// mobject-collections/_Internal/Events/Collection/CollectionEvent
{attribute 'linkalways'} 
{attribute 'no_explicit_call' := 'This FB is a CLASS and must be accessed using methods or properties'}
{attribute 'enable_dynamic_creation'}
FUNCTION_BLOCK ABSTRACT CollectionEvent EXTENDS Disposable
VAR
	_target : I_Collection;
END_VAR

METHOD FB_init : BOOL
VAR_INPUT
	bInitRetains : BOOL; // if TRUE, the retain variables are initialized (warm start / cold start)
	bInCopyCode : BOOL;  // if TRUE, the instance afterwards gets moved into the copy code (online change)
	Target : I_Collection;
END_VAR
This^._target := Target;
END_METHOD

PROPERTY PUBLIC Target : I_Collection
GET
PUBLIC
Target := _target;
END_GET
END_PROPERTY

END_FUNCTION_BLOCK

// mobject-collections/Interfaces/Collections/Events/I_CollectionChangedEvent
INTERFACE I_CollectionChangedEvent EXTENDS I_Event

PROPERTY PUBLIC Target : I_Collection
GET
END_GET
END_PROPERTY

END_INTERFACE

// mobject-collections/_Internal/Events/Collection/CollectionDisposedEvent
{attribute 'linkalways'} 
{attribute 'no_explicit_call' := 'This FB is a CLASS and must be accessed using methods or properties'}
{attribute 'enable_dynamic_creation'}
FUNCTION_BLOCK CollectionDisposedEvent EXTENDS CollectionEvent IMPLEMENTS I_CollectionDisposedEvent

END_FUNCTION_BLOCK

// mobject-collections/Interfaces/Collections/Events/I_CollectionDisposedEvent
INTERFACE I_CollectionDisposedEvent EXTENDS I_Event

PROPERTY PUBLIC Target : I_Collection
GET
END_GET
END_PROPERTY

END_INTERFACE

// mobject-collections/_Internal/Events/KeyValueCollection/KeyValueCollectionChangedEvent
{attribute 'linkalways'} 
{attribute 'no_explicit_call' := 'This FB is a CLASS and must be accessed using methods or properties'}
{attribute 'enable_dynamic_creation'}
FUNCTION_BLOCK KeyValueCollectionChangedEvent EXTENDS KeyValueCollectionEvent IMPLEMENTS I_KeyValueCollectionChangedEvent

END_FUNCTION_BLOCK

// mobject-collections/_Internal/Events/KeyValueCollection/KeyValueCollectionEvent
{attribute 'linkalways'} 
{attribute 'no_explicit_call' := 'This FB is a CLASS and must be accessed using methods or properties'}
{attribute 'enable_dynamic_creation'}
FUNCTION_BLOCK ABSTRACT KeyValueCollectionEvent EXTENDS Disposable
VAR
	_target : I_KeyValueCollection;
END_VAR

METHOD FB_init : BOOL
VAR_INPUT
	bInitRetains : BOOL; // if TRUE, the retain variables are initialized (warm start / cold start)
	bInCopyCode : BOOL;  // if TRUE, the instance afterwards gets moved into the copy code (online change)
	Target : I_KeyValueCollection;
END_VAR
This^._target := Target;
END_METHOD

PROPERTY PUBLIC Target : I_KeyValueCollection
GET
PUBLIC
Target := _target;
END_GET
END_PROPERTY

END_FUNCTION_BLOCK

// mobject-collections/_Internal/Events/KeyValueCollection/KeyValueCollectionDisposedEvent
{attribute 'linkalways'} 
{attribute 'no_explicit_call' := 'This FB is a CLASS and must be accessed using methods or properties'}
{attribute 'enable_dynamic_creation'}
FUNCTION_BLOCK KeyValueCollectionDisposedEvent EXTENDS KeyValueCollectionEvent IMPLEMENTS I_KeyValueCollectionDisposedEvent

END_FUNCTION_BLOCK

// mobject-collections/_Internal/LinkedList/Enumerator/LinkedListForwardEnumerator
{attribute 'linkalways'} 
{attribute 'no_explicit_call' := 'This FB is a CLASS and must be accessed using methods or properties'}
{attribute 'enable_dynamic_creation'}
FUNCTION_BLOCK LinkedListForwardEnumerator EXTENDS Disposable IMPLEMENTS I_ForwardEnumerator, I_EventHandler
VAR
	parent : I_LinkedList;
	currentNode : I_LinkedListNode;
	moveNextCalled : BOOL := FALSE;
	invalid : BOOL := FALSE; 
END_VAR

METHOD FB_init : BOOL
VAR_INPUT
	bInitRetains : BOOL; // if TRUE, the retain variables are initialized (warm start / cold start)
	bInCopyCode : BOOL;  // if TRUE, the instance afterwards gets moved into the copy code (online change)
	Parent : I_LinkedList;
END_VAR
Parent.OnEvent('OnChanged',THIS^);
Parent.OnEvent('OnDisposed',THIS^);
this^.parent := Parent;
END_METHOD

METHOD FB_exit : BOOL
VAR_INPUT
	bInCopyCode : BOOL; // if TRUE, the exit method is called for exiting an instance that is copied afterwards (online change).
END_VAR
IF bInCopyCode THEN
	RETURN;
END_IF

IF parent = 0 THEN
	RETURN;
END_IF

parent.OffEvent('OnChanged',THIS^);
parent.OffEvent('OnDisposed',THIS^);
END_METHOD

METHOD PUBLIC HandleEvent
VAR_INPUT
	Event : I_Event;
END_VAR
VAR
	changedEvent : I_CollectionChangedEvent;
	disposedEvent : I_CollectionDisposedEvent;
END_VAR
IF __QUERYINTERFACE(Event, changedEvent) THEN
	invalid := TRUE;
	currentNode := 0;
ELSIF __QUERYINTERFACE(Event, disposedEvent) THEN
	parent := 0;
	Dispose();
END_IF
END_METHOD

PROPERTY PUBLIC IsValid : BOOL
GET
PUBLIC
IsValid := (not invalid and parent <> 0);
END_GET
END_PROPERTY

METHOD PUBLIC MoveNext : BOOL
IF invalid THEN
	RETURN;
END_IF

IF NOT moveNextCalled THEN
	moveNextCalled := TRUE;	
	currentNode := parent.First;
	MoveNext := currentNode <> 0;
	RETURN;
END_IF

IF currentNode = 0 THEN
	RETURN;
END_IF

if currentNode.Next <> 0 then
	currentNode := currentNode.Next;
	MoveNext := TRUE;	
	RETURN;
END_IF
END_METHOD

METHOD Reset
VAR_INPUT
END_VAR
moveNextCalled := FALSE;
currentNode := 0;
END_METHOD

METHOD PUBLIC TryGet : BOOL;
VAR_INPUT
	Destination : ANY;
END_VAR
IF currentNode <> 0 THEN
	TryGet := currentNode.TryGet(Destination);
END_IF
END_METHOD

METHOD PUBLIC TryGetTo : BOOL;
VAR_INPUT
	DestinationAddress : PVOID;
	DestinationSize : UDINT;
END_VAR
IF currentNode <> 0 THEN
	TryGetTo := currentNode.TryGetTo(DestinationAddress,DestinationSize);
END_IF
END_METHOD

END_FUNCTION_BLOCK

// mobject-collections/Interfaces/Collections/I_LinkedList
INTERFACE I_LinkedList EXTENDS I_Collection

METHOD PUBLIC AddAfter
VAR_INPUT
	After : I_LinkedListNode;
	Value : ANY;
END_VAR
END_METHOD

METHOD PUBLIC AddBefore
VAR_INPUT
	Before : I_LinkedListNode;
	Value : ANY;
END_VAR
END_METHOD

METHOD PUBLIC AddFirst
VAR_INPUT
	Value : ANY;
END_VAR
END_METHOD

METHOD PUBLIC AddLast
VAR_INPUT
	Value : ANY;
END_VAR
END_METHOD

METHOD PUBLIC Find : I_LinkedListNode
VAR_INPUT
	Value : ANY;
END_VAR
END_METHOD

METHOD PUBLIC FindLast : I_LinkedListNode
VAR_INPUT
	Value : ANY;
END_VAR
END_METHOD

PROPERTY PUBLIC First : I_LinkedListNode
GET
END_GET
END_PROPERTY

PROPERTY PUBLIC Last : I_LinkedListNode
GET
END_GET
END_PROPERTY

METHOD PUBLIC Remove
VAR_INPUT
	Value : ANY;
END_VAR
END_METHOD

METHOD PUBLIC RemoveFirst
END_METHOD

METHOD PUBLIC RemoveLast
END_METHOD

END_INTERFACE

// mobject-collections/Interfaces/Collections/Nodes/I_LinkedListNode
INTERFACE I_LinkedListNode EXTENDS I_CollectionNode

PROPERTY PUBLIC Next : I_LinkedListNode
GET
END_GET
SET
END_SET
END_PROPERTY

PROPERTY PUBLIC Previous : I_LinkedListNode
GET
END_GET
SET
END_SET
END_PROPERTY

END_INTERFACE

// mobject-collections/_Internal/LinkedList/Node/LinkedListNode
{attribute 'linkalways'} 
{attribute 'no_explicit_call' := 'This FB is a CLASS and must be accessed using methods or properties'}
{attribute 'enable_dynamic_creation'}
FUNCTION_BLOCK LinkedListNode EXTENDS Disposable IMPLEMENTS I_LinkedListNode
VAR
	pBuffer : POINTER TO BYTE;
	bufferSize : UDINT;
	_previous : I_LinkedListNode;
	_next : I_LinkedListNode;
END_VAR

METHOD FB_init : BOOL
VAR_INPUT
	bInitRetains : BOOL; // if TRUE, the retain variables are initialized (warm start / cold start)
	bInCopyCode : BOOL;  // if TRUE, the instance afterwards gets moved into the copy code (online change)
	Source : ANY;
END_VAR
CreateBuffer(DINT_TO_UDINT(Source.diSize));
CopySourceToBuffer(Source.pValue);
END_METHOD

METHOD FB_exit : BOOL
VAR_INPUT
	bInCopyCode : BOOL; // if TRUE, the exit method is called for exiting an instance that is copied afterwards (online change).
END_VAR
IF bInCopyCode THEN
	RETURN;
END_IF

DestroyBuffer();
END_METHOD

METHOD PRIVATE CopyBufferToDestination
VAR_INPUT
	DestinationAddress : PVOID;
END_VAR
MEMCPY(DestinationAddress, pBuffer, bufferSize);
END_METHOD

METHOD PRIVATE CopySourceToBuffer
VAR_INPUT
	SourceAddress : PVOID;
END_VAR
MEMCPY(pBuffer, SourceAddress, bufferSize);
END_METHOD

METHOD PRIVATE CreateBuffer
VAR_INPUT
	SizeInBytes : UDINT;
END_VAR
bufferSize := SizeInBytes;
pBuffer := __NEW(BYTE, SizeInBytes);
END_METHOD

METHOD PRIVATE DestroyBuffer
IF pBuffer = 0 THEN
	RETURN;
END_IF

__DELETE(pBuffer);
bufferSize := 0;
END_METHOD

PROPERTY PUBLIC DataSize : UDINT
GET
PUBLIC
DataSize := bufferSize;
END_GET
END_PROPERTY

METHOD PUBLIC Equals : BOOL
VAR_INPUT
	Symbol : ANY;
END_VAR
IF pBuffer = 0 THEN
	RETURN;
END_IF

IF bufferSize <> DINT_TO_UDINT(Symbol.diSize) THEN
	RETURN;
END_IF

Equals := MEMCMP(Symbol.pValue, pBuffer, bufferSize) = 0;
END_METHOD

PROPERTY PUBLIC Next : I_LinkedListNode
GET
PUBLIC
Next := _next;
END_GET
SET
PUBLIC
_next := Next;
END_SET
END_PROPERTY

PROPERTY PUBLIC Previous : I_LinkedListNode
GET
PUBLIC
Previous := _previous;
END_GET
SET
PUBLIC
_previous := Previous;
END_SET
END_PROPERTY

METHOD PUBLIC TryGet : BOOL;
VAR_INPUT
	Destination : ANY;
END_VAR
TryGet := TryGetTo(Destination.pValue, DINT_TO_UDINT(Destination.diSize));
END_METHOD

METHOD PUBLIC TryGetTo : BOOL;
VAR_INPUT
	DestinationAddress : PVOID;
	DestinationSize : UDINT;
END_VAR
IF pBuffer = 0 THEN
	RETURN;
END_IF

IF bufferSize <> DestinationSize THEN
	RETURN;
END_IF

CopyBufferToDestination(DestinationAddress);
TryGetTo := TRUE;
END_METHOD

END_FUNCTION_BLOCK

// mobject-collections/_Internal/OrderedDictionary/Enumerator/OrderedDictionaryForwardEnumerator
{attribute 'linkalways'} 
{attribute 'no_explicit_call' := 'This FB is a CLASS and must be accessed using methods or properties'}
{attribute 'enable_dynamic_creation'}
FUNCTION_BLOCK OrderedDictionaryForwardEnumerator EXTENDS Disposable IMPLEMENTS I_KeyValueForwardEnumerator, I_EventHandler
VAR
	parent : I_Dictionary;
	nodes : I_Collection;
	collectionEnumerator : I_ForwardEnumerator;
	currentNode : I_OrderedDictionaryTreeNode;
	moveNextCalled : BOOL := FALSE;
	invalid : BOOL := FALSE; 
END_VAR

METHOD FB_init : BOOL
VAR_INPUT
	bInitRetains : BOOL; // if TRUE, the retain variables are initialized (warm start / cold start)
	bInCopyCode : BOOL;  // if TRUE, the instance afterwards gets moved into the copy code (online change)
	Parent : I_Dictionary;
	Nodes : I_Collection;
END_VAR
Parent.OnEvent('OnChanged',THIS^);
Parent.OnEvent('OnDisposed',THIS^);
THIS^.parent := Parent;
THIS^.nodes := Nodes;
THIS^.collectionEnumerator := Nodes.GetEnumerator();
END_METHOD

METHOD FB_exit : BOOL
VAR_INPUT
	bInCopyCode : BOOL; // if TRUE, the exit method is called for exiting an instance that is copied afterwards (online change).
END_VAR
IF bInCopyCode THEN
	RETURN;
END_IF

collectionEnumerator.Dispose();
nodes.Dispose();

IF parent = 0 THEN
	RETURN;
END_IF

parent.OffEvent('OnChanged',THIS^);
parent.OffEvent('OnDisposed',THIS^);
END_METHOD

METHOD PUBLIC HandleEvent
VAR_INPUT
	Event : I_Event;
END_VAR
VAR
	changedEvent : I_KeyValueCollectionChangedEvent;
	disposedEvent : I_KeyValueCollectionDisposedEvent;
END_VAR
IF __QUERYINTERFACE(Event, changedEvent) THEN
	invalid := TRUE;
	currentNode := 0;
ELSIF __QUERYINTERFACE(Event, disposedEvent) THEN
	parent := 0;	
	Dispose();
END_IF
END_METHOD

PROPERTY PUBLIC IsValid : BOOL
GET
PUBLIC
IsValid := (not invalid and parent <> 0);
END_GET
END_PROPERTY

PROPERTY PUBLIC Key : T_MAXSTRING
GET
IF NOT IsValid THEN
	RETURN;
END_IF

IF currentNode = 0 THEN
	RETURN;
END_IF

Key := currentNode.Key;
END_GET
END_PROPERTY

METHOD PUBLIC MoveNext : BOOL
IF invalid THEN
	RETURN;
END_IF

IF collectionEnumerator.MoveNext() THEN
	collectionEnumerator.TryGet(currentNode);
	MoveNext := TRUE;
END_IF
END_METHOD

METHOD Reset
VAR_INPUT
END_VAR
moveNextCalled := FALSE;
collectionEnumerator.Reset();
END_METHOD

METHOD PUBLIC TryGet : BOOL;
VAR_INPUT
	Destination : ANY;
END_VAR
IF currentNode <> 0 THEN
	TryGet := currentNode.TryGet(Destination);
END_IF
END_METHOD

METHOD PUBLIC TryGetTo : BOOL;
VAR_INPUT
	DestinationAddress : PVOID;
	DestinationSize : UDINT;
END_VAR
IF currentNode <> 0 THEN
	TryGetTo := currentNode.TryGetTo(DestinationAddress,DestinationSize);
END_IF
END_METHOD

END_FUNCTION_BLOCK

// mobject-collections/Interfaces/KeyValueCollections/Nodes/I_OrderedDictionaryTreeNode
INTERFACE I_OrderedDictionaryTreeNode EXTENDS I_CollectionNode

METHOD PUBLIC DeepCopy
VAR_INPUT
	Node : I_OrderedDictionaryTreeNode;
END_VAR
END_METHOD

PROPERTY PUBLIC Height : DINT
GET
END_GET
SET
END_SET
END_PROPERTY

PROPERTY PUBLIC Key : T_MAXSTRING
GET
END_GET
END_PROPERTY

PROPERTY PUBLIC Left : I_OrderedDictionaryTreeNode
GET
END_GET
SET
END_SET
END_PROPERTY

PROPERTY PUBLIC Next : I_OrderedDictionaryTreeNode
GET
END_GET
SET
END_SET
END_PROPERTY

PROPERTY PUBLIC NodeBufferPointer : Pointer To Byte
GET
END_GET
END_PROPERTY

PROPERTY PUBLIC NodeBufferSize : UDINT
GET
END_GET
END_PROPERTY

PROPERTY PUBLIC Previous : I_OrderedDictionaryTreeNode
GET
END_GET
SET
END_SET
END_PROPERTY

METHOD Reinitialize
VAR_INPUT
	Key : T_MAXSTRING;
	Source : ANY;
END_VAR
END_METHOD

PROPERTY PUBLIC Right : I_OrderedDictionaryTreeNode
GET
END_GET
SET
END_SET
END_PROPERTY

END_INTERFACE

// mobject-collections/_Internal/OrderedDictionary/Node/OrderedDictionaryTreeNode
{attribute 'linkalways'} 
{attribute 'no_explicit_call' := 'This FB is a CLASS and must be accessed using methods or properties'}
{attribute 'enable_dynamic_creation'}
FUNCTION_BLOCK OrderedDictionaryTreeNode EXTENDS Disposable IMPLEMENTS I_OrderedDictionaryTreeNode
VAR
	_key : T_MAXSTRING;
	pBuffer : POINTER TO BYTE;
	bufferSize : UDINT;
    _height : DINT;
    _left : I_OrderedDictionaryTreeNode;
    _right : I_OrderedDictionaryTreeNode;
	_next : I_OrderedDictionaryTreeNode;
    _previous : I_OrderedDictionaryTreeNode;
END_VAR

METHOD FB_init : BOOL
VAR_INPUT
	bInitRetains : BOOL; // if TRUE, the retain variables are initialized (warm start / cold start)
	bInCopyCode : BOOL;  // if TRUE, the instance afterwards gets moved into the copy code (online change)
	NodeKey : T_MAXSTRING;
	NodeSource : ANY;
END_VAR
_key := NodeKey;
CreateBuffer(DINT_TO_UDINT(NodeSource.diSize));
CopySourceToBuffer(NodeSource.pValue);
END_METHOD

METHOD FB_exit : BOOL
VAR_INPUT
	bInCopyCode : BOOL; // if TRUE, the exit method is called for exiting an instance that is copied afterwards (online change).
END_VAR
IF bInCopyCode THEN
	RETURN;
END_IF

DestroyBuffer();
END_METHOD

METHOD PRIVATE CopyBufferToDestination
VAR_INPUT
	DestinationAddress : PVOID;
END_VAR
MEMCPY(DestinationAddress, pBuffer, bufferSize);
END_METHOD

METHOD PRIVATE CopySourceToBuffer
VAR_INPUT
	SourceAddress : PVOID;
END_VAR
MEMCPY(pBuffer, SourceAddress, bufferSize);
END_METHOD

METHOD PRIVATE CreateBuffer
VAR_INPUT
	SizeInBytes : UDINT;
END_VAR
bufferSize := SizeInBytes;
pBuffer := __NEW(BYTE, SizeInBytes);
END_METHOD

METHOD PRIVATE DestroyBuffer
VAR_INPUT
END_VAR
IF pBuffer = 0 THEN
	RETURN;
END_IF

__DELETE(pBuffer);
bufferSize := 0;
END_METHOD

PROPERTY PUBLIC DataSize : UDINT
GET
DataSize := bufferSize;
END_GET
END_PROPERTY

METHOD PUBLIC DeepCopy
VAR_INPUT
	Node : I_OrderedDictionaryTreeNode;
END_VAR
DestroyBuffer();
CreateBuffer(Node.NodeBufferSize);
CopySourceToBuffer(Node.NodeBufferPointer);
_key := Node.Key;
_previous := Node.Previous;
_next := Node.Next;
END_METHOD

METHOD PUBLIC Equals : BOOL
VAR_INPUT
	Symbol : ANY;
END_VAR
IF pBuffer = 0 THEN
	RETURN;
END_IF

IF bufferSize <> DINT_TO_UDINT(symbol.diSize) THEN
	RETURN;
END_IF

Equals := MEMCMP(Symbol.pValue, pBuffer, bufferSize) = 0;
END_METHOD

PROPERTY PUBLIC Height : DINT
GET
Height := _height;
END_GET
SET
PUBLIC 
VAR
END_VAR
_height := Height;
END_SET
END_PROPERTY

PROPERTY PUBLIC Key : T_MAXSTRING
GET
Key := _key;
END_GET
END_PROPERTY

PROPERTY PUBLIC Left : I_OrderedDictionaryTreeNode
GET
Left := _left;
END_GET
SET
_left := Left;
END_SET
END_PROPERTY

PROPERTY PUBLIC Next : I_OrderedDictionaryTreeNode
GET
Next := _next;
END_GET
SET
_next := Next;
END_SET
END_PROPERTY

PROPERTY PUBLIC NodeBufferPointer : Pointer To Byte
GET
NodeBufferPointer := pBuffer;
END_GET
END_PROPERTY

PROPERTY PUBLIC NodeBufferSize : UDINT
GET
NodeBufferSize := bufferSize;
END_GET
END_PROPERTY

PROPERTY PUBLIC Previous : I_OrderedDictionaryTreeNode
GET
Previous := _previous;
END_GET
SET
_previous := Previous;
END_SET
END_PROPERTY

METHOD Reinitialize
VAR_INPUT
	Key : T_MAXSTRING;
	Source : ANY;
END_VAR
_key := Key;

IF pBuffer <> 0 THEN
	DestroyBuffer();
END_IF

CreateBuffer(DINT_TO_UDINT(Source.diSize));
CopySourceToBuffer(Source.pValue);
END_METHOD

PROPERTY PUBLIC Right : I_OrderedDictionaryTreeNode
GET
Right := _right;
END_GET
SET
_right := Right;
END_SET
END_PROPERTY

METHOD TryGet : BOOL
VAR_INPUT
	Destination	: ANY;
END_VAR
TryGet := TryGetTo(Destination.pValue, DINT_TO_UDINT(Destination.diSize));
END_METHOD

METHOD TryGetTo : BOOL
VAR_INPUT
	DestinationAddress : PVOID;
	DestinationSize : UDINT;
END_VAR
IF pBuffer = 0 THEN
	RETURN;
END_IF

IF bufferSize <> DestinationSize THEN
	RETURN;
END_IF

CopyBufferToDestination(DestinationAddress);
TryGetTo := TRUE;
END_METHOD

END_FUNCTION_BLOCK

// mobject-collections/Dictionary/Dictionary
{attribute 'linkalways'} 
{attribute 'no_explicit_call' := 'This FB is a CLASS and must be accessed using methods or properties'}
{attribute 'enable_dynamic_creation'}
FUNCTION_BLOCK Dictionary EXTENDS Disposable IMPLEMENTS I_Dictionary
VAR
	eventEmitter : EventEmitter;
	rootNode : I_DictionaryTreeNode;
END_VAR

METHOD FB_exit : BOOL
VAR_INPUT
	bInCopyCode : BOOL; // if TRUE, the exit method is called for exiting an instance that is copied afterwards (online change).
END_VAR
VAR
END_VAR
IF bInCopyCode THEN
    RETURN;
END_IF

Clear();
EmitDisposedEvent();
END_METHOD

METHOD PRIVATE Balance : I_DictionaryTreeNode
VAR_INPUT
	Node : I_DictionaryTreeNode;
END_VAR
VAR
	balanceFactor : DINT;
END_VAR
balanceFactor := THIS^.GetBalanceFactor(Node);

IF (balanceFactor > 1) THEN
	IF THIS^.GetBalanceFactor(Node.Left) < 0 THEN
		Node.Left := THIS^.LeftRotate(Node.Left);
	END_IF
	Node := RightRotate(Node);
ELSIF (balanceFactor < -1) THEN
	IF THIS^.GetBalanceFactor(Node.Right) > 0 THEN
		Node.Right := RightRotate(Node.Right);
	END_IF
	Node := LeftRotate(Node);
END_IF

Balance := Node;
END_METHOD

METHOD PRIVATE EmitChangedEvent
VAR
	pDictionaryChangedEvent : POINTER TO KeyValueCollectionChangedEvent;
END_VAR
pDictionaryChangedEvent := __NEW(KeyValueCollectionChangedEvent(Target := THIS^));
eventEmitter.Emit('OnChanged', pDictionaryChangedEvent^);
pDictionaryChangedEvent^.Dispose();
END_METHOD

METHOD PRIVATE EmitDisposedEvent
VAR
	pDictionaryDisposedEvent : POINTER TO KeyValueCollectionDisposedEvent;
END_VAR
pDictionaryDisposedEvent := __NEW(KeyValueCollectionDisposedEvent(Target := THIS^));
eventEmitter.Emit('OnDisposed', pDictionaryDisposedEvent^);
pDictionaryDisposedEvent^.Dispose();
END_METHOD

METHOD PRIVATE FindMinimum : I_DictionaryTreeNode
VAR_INPUT
	Node : I_DictionaryTreeNode;
END_VAR
VAR
	nextNode : I_DictionaryTreeNode;
END_VAR
nextNode := Node;

WHILE (nextNode.left <> 0) DO
      nextNode := nextNode.left;
END_WHILE;

FindMinimum := nextNode;
END_METHOD

METHOD PRIVATE GetBalanceFactor : DINT
VAR_INPUT
	Node : I_DictionaryTreeNode;
END_VAR
IF (Node = 0) THEN
	GetBalanceFactor := 0;
	RETURN;
END_IF

GetBalanceFactor := THIS^.GetHeight(node.left) - THIS^.GetHeight(node.right);
END_METHOD

METHOD PRIVATE GetHeight : DINT
VAR_INPUT
	Node : I_DictionaryTreeNode;
END_VAR
IF Node = 0 THEN
	GetHeight := -1;
	RETURN;
END_IF

GetHeight := Node.Height;
END_METHOD

METHOD PRIVATE LeftRotate : I_DictionaryTreeNode
VAR_INPUT
	X : I_DictionaryTreeNode;
END_VAR
VAR
	y : I_DictionaryTreeNode;
	t2 : I_DictionaryTreeNode;
END_VAR
y := X.right;
t2 := y.left;
y.left := X;
X.right := t2;
THIS^.UpdateHeight(X);
THIS^.UpdateHeight(y);
LeftRotate := y;
END_METHOD

METHOD PRIVATE RecursiveAddKeysInOrderToCollection
VAR_INPUT
	Node : I_DictionaryTreeNode;
	Collection : I_Collection;
END_VAR
VAR
	key : T_MAXSTRING;
END_VAR
IF Node = 0 THEN
	RETURN;
END_IF

THIS^.RecursiveAddKeysInOrderToCollection(Node.Left,Collection);
key := Node.Key;
Collection.AddItem(key);
THIS^.RecursiveAddKeysInOrderToCollection(Node.Right,Collection);
END_METHOD

METHOD PRIVATE RecursiveAddNodesInOrderToCollection
VAR_INPUT
	Node : I_DictionaryTreeNode;
	Collection : I_Collection;
END_VAR
IF Node = 0 THEN
	RETURN;
END_IF

THIS^.RecursiveAddNodesInOrderToCollection(Node.Left,Collection);
Collection.AddItem(Node);
THIS^.RecursiveAddNodesInOrderToCollection(Node.Right,Collection);
END_METHOD

METHOD PRIVATE RecursiveClear
VAR_INPUT
	Node : I_DictionaryTreeNode;
END_VAR
VAR
	thisNodeKey : T_MAXSTRING;
	leftNodeKey : T_MAXSTRING;
	rightNodeKey : T_MAXSTRING;
END_VAR
IF (Node = 0) THEN
	RETURN;
END_IF

thisNodeKey := Node.key;

IF (Node.Left <> 0) THEN
	leftNodeKey := Node.Left.key;
END_IF

IF (Node.Right <> 0) THEN
	rightNodeKey := Node.Right.key;
END_IF


RecursiveClear(Node.Left);
RecursiveClear(Node.Right);
Node.Dispose();
END_METHOD

METHOD PRIVATE RecursiveCountNodes
VAR_INPUT
	Node : I_DictionaryTreeNode;
	Count : REFERENCE TO DINT;
END_VAR
IF Node = 0 THEN
	RETURN;
END_IF

Count := Count + 1;

THIS^.RecursiveCountNodes(Node.Left,Count);
THIS^.RecursiveCountNodes(Node.Right,Count);
END_METHOD

METHOD PRIVATE RecursiveDelete : I_DictionaryTreeNode
VAR_INPUT
	Key : T_MAXSTRING;
	Node : I_DictionaryTreeNode;
END_VAR
VAR
	newNode : I_DictionaryTreeNode; 
	minValueNode : I_DictionaryTreeNode;
	minValueNodeParent : I_DictionaryTreeNode;
	balanceFactor : DINT;
END_VAR
IF (Node = 0) THEN
    RETURN;
END_IF

IF (Key < Node.Key) THEN
    Node.left := THIS^.RecursiveDelete(Key, Node.left);
ELSIF (Key > Node.Key) THEN
    Node.right := THIS^.RecursiveDelete(Key, Node.right);
ELSE
    IF (Node.Left = 0) OR (Node.Right = 0) THEN
        IF (Node.Left = 0) THEN
            newNode := Node.Right;
        ELSE
            newNode := Node.Left;
        END_IF

        Node.Dispose();
        THIS^.updateHeight(newNode);
        RecursiveDelete := THIS^.Balance(newNode);
        RETURN;
    ELSE
        minValueNode := FindMinimum(Node.Right);
        Node.DeepCopy(minValueNode);
        Node.Right := THIS^.RecursiveDelete(minValueNode.Key, Node.Right);	
    END_IF
END_IF

THIS^.updateHeight(Node);
RecursiveDelete := THIS^.Balance(Node);
END_METHOD

METHOD PRIVATE RecursiveFind : I_DictionaryTreeNode
VAR_INPUT
	Key : T_MAXSTRING;
	Node : I_DictionaryTreeNode;
END_VAR
IF (Node = 0) THEN
	RETURN;
END_IF

IF (Key < Node.key) THEN
  RecursiveFind := THIS^.RecursiveFind(key, Node.left);
  RETURN;
ELSIF (key > Node.key) THEN
  RecursiveFind := THIS^.RecursiveFind(key, Node.right);
  RETURN;
ELSE 
  RecursiveFind := Node;
  RETURN;
END_IF
END_METHOD

METHOD PRIVATE RecursiveInsert : I_DictionaryTreeNode
VAR_INPUT
	Key : T_MAXSTRING;
	Value : ANY;
	Node : I_DictionaryTreeNode;
END_VAR
VAR
	pAVLTreeNode : POINTER TO DictionaryTreeNode;
	balanceFactor : DINT;
END_VAR
IF (Node = 0) THEN
	pAVLTreeNode := __NEW(DictionaryTreeNode(NodeKey := Key, NodeSource := Value));
	RecursiveInsert := pAVLTreeNode^;
	RETURN;
END_IF

IF (Key < Node.Key) THEN
	Node.left := THIS^.RecursiveInsert(Key, Value, Node.left);
ELSIF (Key > Node.Key) THEN
	Node.right := THIS^.RecursiveInsert(Key, Value, Node.right);
ELSE
	Node.Reinitialize(Key,Value);
	RecursiveInsert := Node;
END_IF

THIS^.updateHeight(node);

Node := balance(Node);
RecursiveInsert := Node;
END_METHOD

METHOD PRIVATE RightRotate : I_DictionaryTreeNode
VAR_INPUT
	Y : I_DictionaryTreeNode;
END_VAR
VAR
	x : I_DictionaryTreeNode;
	t2 : I_DictionaryTreeNode;
END_VAR
x := Y.left;
t2 := x.right;
x.right := Y;
Y.left := t2;
THIS^.UpdateHeight(Y);
THIS^.UpdateHeight(x);
RightRotate := x;
END_METHOD

METHOD PRIVATE UpdateHeight
VAR_INPUT
	Node : I_DictionaryTreeNode;
END_VAR
IF (Node = 0) THEN
	RETURN;
END_IF

Node.height := 1 + MAX(THIS^.GetHeight(Node.left), THIS^.GetHeight(Node.right));
END_METHOD

METHOD PUBLIC AddOrUpdate
VAR_INPUT
	Key : T_MAXSTRING;
	Value : ANY;
END_VAR
rootNode := THIS^.RecursiveInsert(Key, Value, rootNode);
EmitChangedEvent();
END_METHOD

METHOD PUBLIC Clear
VAR_INPUT
END_VAR
IF rootNode = 0 THEN
	RETURN;
END_IF

THIS^.RecursiveClear(rootNode);
rootNode := 0;
EmitChangedEvent();
END_METHOD

METHOD PUBLIC ContainsKey : BOOL
VAR_INPUT
	Key : T_MAXSTRING;
END_VAR
VAR
	foundNode : I_DictionaryTreeNode;
END_VAR
foundNode := THIS^.RecursiveFind(Key, rootNode);

IF foundNode = 0 THEN
	RETURN;
END_IF

ContainsKey := TRUE;
END_METHOD

PROPERTY PUBLIC Count : DINT
GET
VAR
	NodeCount : DINT;
END_VAR
RecursiveCountNodes(rootNode, NodeCount);
Count := NodeCount;
END_GET
END_PROPERTY

METHOD GetEnumerator : I_ForwardEnumerator
VAR
	pNodeCollection : POINTER TO LinkedList;
	pEnumerator : POINTER TO DictionaryForwardEnumerator;
END_VAR
pNodeCollection := __NEW(LinkedList);
THIS^.RecursiveAddNodesInOrderToCollection(rootNode, pNodeCollection^);

pEnumerator := __NEW(DictionaryForwardEnumerator(Parent := THIS^, Nodes := pNodeCollection^));
GetEnumerator := pEnumerator^;
END_METHOD

METHOD PUBLIC GetKeys : I_Collection
VAR
	pLinkedList : POINTER TO LinkedList;
END_VAR
pLinkedList := __NEW(LinkedList);
THIS^.RecursiveAddKeysInOrderToCollection(rootNode,pLinkedList^);
GetKeys := pLinkedList^;
END_METHOD

METHOD GetKeyValueEnumerator : I_KeyValueForwardEnumerator
VAR
	pNodeCollection : POINTER TO LinkedList;
	pEnumerator : POINTER TO DictionaryForwardEnumerator;
END_VAR
pNodeCollection := __NEW(LinkedList);
THIS^.RecursiveAddNodesInOrderToCollection(rootNode, pNodeCollection^);

pEnumerator := __NEW(DictionaryForwardEnumerator(Parent := THIS^, Nodes := pNodeCollection^));
GetKeyValueEnumerator := pEnumerator^;
END_METHOD

PROPERTY IsEmpty : BOOL
GET
IsEmpty := rootNode = 0;
END_GET
END_PROPERTY

METHOD PUBLIC OffEvent
VAR_INPUT
	EventName : T_MaxString;
	EventHandler : I_EventHandler;
END_VAR
eventEmitter.OffEvent(EventName, EventHandler);
END_METHOD

METHOD PUBLIC OnceEvent
VAR_INPUT
	EventName : T_MaxString;
	EventHandler : I_EventHandler;
END_VAR
eventEmitter.OnceEvent(EventName, EventHandler);
END_METHOD

METHOD PUBLIC OnEvent
VAR_INPUT
	EventName : T_MaxString;
	EventHandler : I_EventHandler;
END_VAR
eventEmitter.OnEvent(EventName, EventHandler);
END_METHOD

METHOD PUBLIC Remove
VAR_INPUT
	Key : T_MAXSTRING;
END_VAR
rootNode := THIS^.RecursiveDelete(Key, rootNode);
EmitChangedEvent();
END_METHOD

METHOD PUBLIC TryAdd : BOOL
VAR_INPUT
	Key : T_MAXSTRING;
	Value : ANY;
END_VAR
IF ContainsKey(Key) THEN
	RETURN;
END_IF
	  
THIS^.AddOrUpdate(Key, Value);
TryAdd := TRUE;
END_METHOD

METHOD PUBLIC TryGetValue : BOOL
VAR_INPUT
	Key : T_MAXSTRING;
	Destination	: ANY;
END_VAR
TryGetValue := TryGetValueTo(Key, Destination.pValue, DINT_TO_UDINT(Destination.diSize));
END_METHOD

METHOD PUBLIC TryGetValueTo : BOOL
VAR_INPUT
	Key : T_MAXSTRING;
	DestinationAddress : PVOID;
	DestinationSize : UDINT;
END_VAR
VAR
	foundNode : I_DictionaryTreeNode;
END_VAR
foundNode := THIS^.RecursiveFind(Key, rootNode);

IF foundNode = 0 THEN
	RETURN;
END_IF

TryGetValueTo := foundNode.TryGetTo(DestinationAddress, DestinationSize);
END_METHOD

END_FUNCTION_BLOCK

// mobject-events/EventEmitter/EventEmitter
{attribute 'linkalways'} 
{attribute 'no_explicit_call' := 'This FB is a CLASS and must be accessed using methods or properties'}
{attribute 'enable_dynamic_creation'}
FUNCTION_BLOCK EventEmitter EXTENDS Disposable IMPLEMENTS I_EventEmitter, I_EventTarget
VAR
	firstEventHandlerItem : I_EventHandlerItem;
END_VAR

METHOD FB_exit : BOOL
VAR_INPUT
	bInCopyCode : BOOL; // if TRUE, the exit method is called for exiting an instance that is copied afterwards (online change).
END_VAR
IF bInCopyCode THEN
	RETURN;
END_IF

DisposeAllEventHandlerItems();
END_METHOD

METHOD PRIVATE DisposeAllEventHandlerItems
VAR_INPUT
END_VAR
WHILE firstEventHandlerItem <> 0 DO
	DisposeEventHandlerItem(firstEventHandlerItem);
END_WHILE
END_METHOD

METHOD PRIVATE DisposeEventHandlerItem
VAR_INPUT
	EventHandlerItem : I_EventHandlerItem;
END_VAR
RemoveEventHandlerItemFromCollection(EventHandlerItem);
EventHandlerItem.Dispose();
END_METHOD

METHOD PRIVATE FindEventHandlerItem : I_EventHandlerItem
VAR_INPUT
	EventName : T_MaxString;
	EventHandler : I_EventHandler;
END_VAR
VAR
	currentEventHandlerItem : I_EventHandlerItem;
END_VAR
currentEventHandlerItem := firstEventHandlerItem;

WHILE currentEventHandlerItem <> 0 DO
	
	IF currentEventHandlerItem.EqualTo(EventName, EventHandler) THEN
		FindEventHandlerItem := currentEventHandlerItem; 
		RETURN;
	END_IF
	
	currentEventHandlerItem := currentEventHandlerItem.Next;

END_WHILE
END_METHOD

METHOD PRIVATE InsertEventHandlerItem
VAR_INPUT
	EventHandlerItem : I_EventHandlerItem;
END_VAR
VAR
	currentEventHandlerItem : I_EventHandlerItem;
END_VAR
IF firstEventHandlerItem = 0 THEN
	firstEventHandlerItem := EventHandlerItem;
	RETURN;
END_IF

currentEventHandlerItem := firstEventHandlerItem;

WHILE currentEventHandlerItem.next <> 0 DO
	currentEventHandlerItem := currentEventHandlerItem.next;
END_WHILE

currentEventHandlerItem.next := EventHandlerItem;
EventHandlerItem.previous := currentEventHandlerItem;
END_METHOD

METHOD PRIVATE RemoveEventHandlerItemFromCollection
VAR_INPUT
	EventHandlerItem : I_EventHandlerItem;
END_VAR
VAR
	previous : I_EventHandlerItem;
	next : I_EventHandlerItem;
END_VAR
IF EventHandlerItem = 0 THEN
	// nothing to remove
	RETURN;
END_IF

IF EventHandlerItem = firstEventHandlerItem AND EventHandlerItem.Next = 0 THEN 
	
	// the item was the only one in the list, as such you just set the first to zero
	firstEventHandlerItem := 0; 
	
ELSIF EventHandlerItem = firstEventHandlerItem THEN 
	
	// the item was the first in the list of many, so make the next item the first and remove 
	// it's "previous" as the first in the item does not have a previous
	firstEventHandlerItem := EventHandlerItem.next; 
	firstEventHandlerItem.Previous := 0;

ELSIF EventHandlerItem.Next <> 0 THEN
	
	// the item is mid list so link it's previous and next together 
	previous := EventHandlerItem.Previous;
	next := EventHandlerItem.Next;
	
	previous.Next := next;
	next.Previous := previous;
	
ELSE 
	
	// the item is at the end so only remove itself from the previous
	previous := EventHandlerItem.Previous;
	previous.Next := 0;

END_IF
END_METHOD

METHOD PUBLIC Clear
VAR_INPUT
END_VAR
DisposeAllEventHandlerItems();
END_METHOD

METHOD PUBLIC Emit
VAR_INPUT
	EventName : T_MaxString;
	Event : I_Event;
END_VAR
VAR
	currentEventHandlerItem : I_EventHandlerItem;
END_VAR
currentEventHandlerItem := firstEventHandlerItem;

WHILE currentEventHandlerItem <> 0 DO
	currentEventHandlerItem.Emit(EventName, Event);
	currentEventHandlerItem := currentEventHandlerItem.Next;
END_WHILE
END_METHOD

METHOD PUBLIC OffEvent
VAR_INPUT
	EventName : T_MaxString;
	EventHandler : I_EventHandler;
END_VAR
VAR
	foundHandlerItem : I_EventHandlerItem;
END_VAR
foundHandlerItem := FindEventHandlerItem(EventName, EventHandler);

IF foundHandlerItem = 0 THEN
	RETURN;
END_IF

DisposeEventHandlerItem(foundHandlerItem);
END_METHOD

METHOD PUBLIC OnceEvent
VAR_INPUT
	EventName : T_MaxString;
	EventHandler : I_EventHandler;
END_VAR
VAR
	pEventHandlerItem : POINTER TO EventHandlerItemOnceOnly;
END_VAR
pEventHandlerItem := __NEW(EventHandlerItemOnceOnly(Name := EventName, Handler := EventHandler, Parent := THIS^));
InsertEventHandlerItem(pEventHandlerItem^);
END_METHOD

METHOD PUBLIC OnEvent
VAR_INPUT
	EventName : T_MaxString;
	EventHandler : I_EventHandler;
END_VAR
VAR
	pEventHandlerItem : POINTER TO EventHandlerItem;
END_VAR
pEventHandlerItem := __NEW(EventHandlerItem(Name :=EventName, Handler := EventHandler));
InsertEventHandlerItem(pEventHandlerItem^);
END_METHOD

END_FUNCTION_BLOCK

// mobject-events/Interfaces/I_EventTarget
INTERFACE I_EventTarget EXTENDS __SYSTEM.IQueryInterface

METHOD PUBLIC Emit
VAR_INPUT
	EventName : T_MaxString;
	Event : I_Event;
END_VAR
END_METHOD

END_INTERFACE

// mobject-events/_Internal/EventHandlerItem/I_EventHandlerItem
INTERFACE I_EventHandlerItem EXTENDS I_Disposable

METHOD PUBLIC Emit : BOOL
VAR_INPUT
	EventName : T_MaxString;
	Event : I_Event;
END_VAR
END_METHOD

METHOD PUBLIC EqualTo : BOOL
VAR_INPUT
	Name : T_MaxString;
	Handler : I_EventHandler;
END_VAR
END_METHOD

PROPERTY PUBLIC Next : I_EventHandlerItem
GET
END_GET
SET
END_SET
END_PROPERTY

PROPERTY PUBLIC Previous : I_EventHandlerItem
GET
END_GET
SET
END_SET
END_PROPERTY

END_INTERFACE

// mobject-events/_Internal/EventHandlerItem/EventHandlerItem
{attribute 'linkalways'} 
{attribute 'no_explicit_call' := 'This FB is a CLASS and must be accessed using methods or properties'}
{attribute 'enable_dynamic_creation'}
FUNCTION_BLOCK EventHandlerItem EXTENDS Disposable IMPLEMENTS I_EventHandlerItem
VAR
	name : T_MAXSTRING;
	handler : I_EventHandler;
	_next : I_EventHandlerItem;
	_previous : I_EventHandlerItem;
END_VAR

METHOD FB_init : BOOL
VAR_INPUT
	bInitRetains : BOOL; // if TRUE, the retain variables are initialized (warm start / cold start)
	bInCopyCode : BOOL;  // if TRUE, the instance afterwards gets moved into the copy code (online change)
	Name : T_MAXSTRING;
	Handler : I_EventHandler;
END_VAR
THIS^.name := Name;
THIS^.handler := Handler;
END_METHOD

METHOD PUBLIC Emit : BOOL
VAR_INPUT
	EventName : T_MaxString;
	Event : I_Event;
END_VAR
IF EventName <> name THEN
	RETURN;
END_IF

IF handler = 0 THEN
	RETURN;
END_IF

handler.HandleEvent(Event);
Emit := TRUE;
END_METHOD

METHOD PUBLIC EqualTo : BOOL
VAR_INPUT
	Name : T_MaxString;
	Handler : I_EventHandler;
END_VAR
IF THIS^.handler <> Handler THEN
	RETURN;
END_IF

IF THIS^.name <> Name THEN
	RETURN;
END_IF

EqualTo := TRUE;
END_METHOD

PROPERTY PUBLIC Next : I_EventHandlerItem
GET
Next := _next;
END_GET
SET
_next := Next;
END_SET
END_PROPERTY

PROPERTY PUBLIC Previous : I_EventHandlerItem
GET
Previous := _previous;
END_GET
SET
_previous := Previous;
END_SET
END_PROPERTY

END_FUNCTION_BLOCK

// mobject-events/_Internal/EventHandlerItem/EventHandlerItemOnceOnly
{attribute 'linkalways'} 
{attribute 'no_explicit_call' := 'This FB is a CLASS and must be accessed using methods or properties'}
{attribute 'enable_dynamic_creation'}
FUNCTION_BLOCK EventHandlerItemOnceOnly EXTENDS EventHandlerItem
VAR
	parent : I_EventEmitter;
END_VAR

METHOD FB_init : BOOL
VAR_INPUT
	bInitRetains : BOOL; // if TRUE, the retain variables are initialized (warm start / cold start)
	bInCopyCode : BOOL;  // if TRUE, the instance afterwards gets moved into the copy code (online change)
	Name : T_MAXSTRING;
	Handler : I_EventHandler;
	Parent : I_EventEmitter;
END_VAR
THIS^.parent := Parent;
END_METHOD

METHOD PUBLIC Emit : BOOL
VAR_INPUT
	EventName : T_MaxString;
	Event : I_Event;
END_VAR
IF NOT SUPER^.Emit(EventName,Event) THEN
	RETURN;
END_IF

parent.OffEvent(name,handler);
Emit := TRUE;
END_METHOD

END_FUNCTION_BLOCK

// mobject-collections/LinkedList/LinkedList
{attribute 'linkalways'} 
{attribute 'no_explicit_call' := 'This FB is a CLASS and must be accessed using methods or properties'}
{attribute 'enable_dynamic_creation'}
FUNCTION_BLOCK LinkedList EXTENDS Disposable IMPLEMENTS I_LinkedList
VAR
	head : I_LinkedListNode;
	tail : I_LinkedListNode;
	eventEmitter : EventEmitter;
END_VAR

METHOD FB_exit : BOOL
VAR_INPUT
	bInCopyCode : BOOL; // if TRUE, the exit method is called for exiting an instance that is copied afterwards (online change).
END_VAR
IF bInCopyCode THEN
	RETURN;
END_IF

Clear();
EmitDisposedEvent();
END_METHOD

METHOD PRIVATE AddNodeAfter
VAR_INPUT
	After : I_LinkedListNode;
	Node : I_LinkedListNode;
END_VAR
VAR
	originalNext : I_LinkedListNode;
END_VAR
IF After = tail THEN
	AddNodeLast(Node);
	RETURN;
END_IF

originalNext := After.Next;
After.Next := Node;
Node.Previous := After;
Node.Next := originalNext;
originalNext.Previous := Node;
END_METHOD

METHOD PRIVATE AddNodeBefore
VAR_INPUT
	Before : I_LinkedListNode;
	Node : I_LinkedListNode;
END_VAR
VAR
	originalBefore : I_LinkedListNode;
END_VAR
IF Before = head THEN
	AddNodeFirst(Node);
	RETURN;
END_IF

originalBefore := Before.Previous;
Before.Previous := Node;
Node.Next := Before;
Node.Previous := originalBefore;
originalBefore.Next := Node;
END_METHOD

METHOD PRIVATE AddNodeFirst
VAR_INPUT
	Node : I_LinkedListNode;
END_VAR
VAR
	originalFirst : I_LinkedListNode;
END_VAR
IF IsEmpty THEN
	head := Node;
	tail := Node; 
	RETURN;	
END_IF

originalFirst := head;
head := Node;
Node.Next := originalFirst;
originalFirst.Previous := Node;
END_METHOD

METHOD PRIVATE AddNodeLast
VAR_INPUT
	Node : I_LinkedListNode;
END_VAR
VAR
	originalLast : I_LinkedListNode;
END_VAR
IF IsEmpty THEN
	head := Node;
	tail := Node; 
	RETURN;	
END_IF

originalLast := tail;
tail := Node;
Node.Previous := originalLast;
originalLast.Next := Node;
END_METHOD

METHOD PRIVATE ContainsLinkedListNode : BOOL
VAR_INPUT
    Node : I_LinkedListNode;
END_VAR
VAR
	current : I_LinkedListNode;
END_VAR
IF IsEmpty THEN	
	RETURN;
END_IF

current := head; 

WHILE current <> 0 DO
	IF current = Node THEN
		ContainsLinkedListNode := TRUE;
		RETURN;
	END_IF
	current := current.next; 
END_WHILE;
END_METHOD

METHOD PRIVATE CreateNode : I_LinkedListNode
VAR_INPUT
	Value : ANY;
END_VAR
VAR
	pLinkedListItem : POINTER TO LinkedListNode;
END_VAR
pLinkedListItem := __NEW(LinkedListNode(Source := Value)); 
CreateNode := pLinkedListItem^;
END_METHOD

METHOD PRIVATE EmitChangedEvent
VAR
	pCollectionChangedEvent : POINTER TO CollectionChangedEvent;
END_VAR
pCollectionChangedEvent := __NEW(CollectionChangedEvent(Target := THIS^));
eventEmitter.Emit('OnChanged', pCollectionChangedEvent^);
pCollectionChangedEvent^.Dispose();
END_METHOD

METHOD PRIVATE EmitDisposedEvent
VAR
	pCollectionDisposedEvent : POINTER TO CollectionDisposedEvent;
END_VAR
pCollectionDisposedEvent := __NEW(CollectionDisposedEvent(Target := THIS^));
eventEmitter.Emit('OnDisposed', pCollectionDisposedEvent^);
pCollectionDisposedEvent^.Dispose();
END_METHOD

METHOD PRIVATE FindFirstNodeWithValue : I_LinkedListNode
VAR_INPUT
	Value : ANY;
END_VAR
VAR
	current : I_LinkedListNode;
END_VAR
IF IsEmpty THEN	
	RETURN;
END_IF

current := head; 

WHILE current <> 0 DO
	IF current.Equals(Value) THEN
		FindFirstNodeWithValue := current;
		RETURN;
	END_IF
	current := current.next; 
END_WHILE;
END_METHOD

METHOD PRIVATE FindLastNodeWithValue : I_LinkedListNode
VAR_INPUT
	Value : ANY;
END_VAR
VAR
	current : I_LinkedListNode;
END_VAR
IF IsEmpty THEN	
	RETURN;
END_IF

current := tail; 

WHILE current <> 0 DO
	IF current.Equals(Value) THEN
		FindLastNodeWithValue := current;
		RETURN;
	END_IF
	current := current.Previous; 
END_WHILE;
END_METHOD

METHOD PRIVATE RemoveAllNodes
WHILE First <> 0 DO
	RemoveNode(First);
END_WHILE
END_METHOD

METHOD PRIVATE RemoveNode : BOOL
VAR_INPUT
	Node : I_LinkedListNode;
END_VAR
IF IsEmpty THEN
	RETURN;
END_IF

IF Node = head AND Node = tail THEN
	// node is the only node
	head := 0;
	tail := 0;
	Node.Dispose();
	RETURN;
	
ELSIF Node = head THEN
	// node is the head
	head := node.Next;
	head.Previous := 0;	
	Node.Dispose();
	RETURN;
	
ELSIF Node = tail THEN
	// node is the tail
	tail := node.Previous;
	tail.Next := 0;	
	Node.Dispose();
	RETURN;
ELSE 
	// node is in the middle
	Node.Previous.Next := Node.Next;
	Node.Next.Previous := Node.Previous;
	Node.Dispose();
	RETURN;
END_IF
END_METHOD

METHOD PUBLIC AddAfter
VAR_INPUT
	After : I_LinkedListNode;
	Value : ANY;
END_VAR
VAR
	node : I_LinkedListNode;
END_VAR
IF NOT ContainsLinkedListNode(After) THEN
	RETURN;
END_IF

node := CreateNode(Value);
AddNodeAfter(After,node);
EmitChangedEvent();
END_METHOD

METHOD PUBLIC AddBefore
VAR_INPUT
	Before : I_LinkedListNode;
	Value : ANY;
END_VAR
VAR
	node : I_LinkedListNode;
END_VAR
IF NOT ContainsLinkedListNode(Before) THEN
	RETURN;
END_IF

node := CreateNode(Value);
AddNodeBefore(Before,node);
EmitChangedEvent();
END_METHOD

METHOD PUBLIC AddFirst
VAR_INPUT
	Value : ANY;
END_VAR
VAR
	node : I_LinkedListNode;
END_VAR
node := CreateNode(Value);
AddNodeFirst(node);
EmitChangedEvent();
END_METHOD

METHOD PUBLIC AddItem
VAR_INPUT
	Item : ANY;
END_VAR
AddLast(Item);
END_METHOD

METHOD PUBLIC AddLast
VAR_INPUT
	Value : ANY;
END_VAR
VAR
	node : I_LinkedListNode;
END_VAR
node := CreateNode(Value);
AddNodeLast(node);
EmitChangedEvent();
END_METHOD

METHOD PUBLIC Clear
IF IsEmpty THEN
	return;
END_IF

RemoveAllNodes();
EmitChangedEvent();
END_METHOD

METHOD PUBLIC Contains : BOOL
VAR_INPUT
    Item : ANY;
END_VAR
VAR
    found : I_LinkedListNode;
END_VAR
found := Find(Item);
Contains := found <> 0;
END_METHOD

PROPERTY PUBLIC Count : DINT
GET
VAR
	current : I_LinkedListNode;
END_VAR
current := First;

WHILE current <> 0 DO
	Count := Count + 1;
	current := current.Next;
END_WHILE
END_GET
END_PROPERTY

METHOD PUBLIC Find : I_LinkedListNode
VAR_INPUT
	Value : ANY;
END_VAR
Find := FindFirstNodeWithValue(Value);
END_METHOD

METHOD PUBLIC FindLast : I_LinkedListNode
VAR_INPUT
	Value : ANY;
END_VAR
FindLast := FindLastNodeWithValue(Value);
END_METHOD

PROPERTY PUBLIC First : I_LinkedListNode
GET
First := head;
END_GET
END_PROPERTY

METHOD PUBLIC GetEnumerator : I_ForwardEnumerator
VAR
	pLinkedListForwardEnumerator : POINTER TO LinkedListForwardEnumerator;
END_VAR
pLinkedListForwardEnumerator := __NEW(LinkedListForwardEnumerator(Parent := THIS^));
GetEnumerator := pLinkedListForwardEnumerator^;
END_METHOD

PROPERTY IsEmpty : BOOL
GET
IsEmpty := head = 0;
END_GET
END_PROPERTY

PROPERTY PUBLIC Last : I_LinkedListNode
GET
Last := tail;
END_GET
END_PROPERTY

METHOD PUBLIC OffEvent
VAR_INPUT
	EventName : T_MaxString;
	EventHandler : I_EventHandler;
END_VAR
eventEmitter.OffEvent(EventName, EventHandler);
END_METHOD

METHOD PUBLIC OnceEvent
VAR_INPUT
	EventName : T_MaxString;
	EventHandler : I_EventHandler;
END_VAR
eventEmitter.OnceEvent(EventName, EventHandler);
END_METHOD

METHOD PUBLIC OnEvent
VAR_INPUT
	EventName : T_MaxString;
	EventHandler : I_EventHandler;
END_VAR
eventEmitter.OnEvent(EventName, EventHandler);
END_METHOD

METHOD PUBLIC Remove
VAR_INPUT
	Value : ANY;
END_VAR
TryRemoveItem(Value);
END_METHOD

METHOD PUBLIC RemoveFirst
IF IsEmpty THEN
	RETURN;
END_IF

RemoveNode(First);
EmitChangedEvent();
END_METHOD

METHOD PUBLIC RemoveLast
IF IsEmpty THEN
	RETURN;
END_IF

RemoveNode(Last);
EmitChangedEvent();
END_METHOD

METHOD PUBLIC TryCopyTo : BOOL
VAR_INPUT
	Destination : ANY;
END_VAR
TryCopyTo := TryCopyToLocation(Destination.pValue, DINT_TO_UDINT(Destination.diSize));
END_METHOD

METHOD PUBLIC TryCopyToLocation : BOOL
VAR_INPUT
	DestinationAddress : PVOID;
	DestinationSize : UDINT;
END_VAR
VAR
	currentNode : I_LinkedListNode;
	requiredDestinationSize : UDINT;
	currentPointer : pvoid;
END_VAR
currentNode := First;

// first pass we check to see what the total size of the list will be.
WHILE currentNode <> 0 DO
	requiredDestinationSize := requiredDestinationSize + currentNode.DataSize;
	currentNode := currentNode.Next;
END_WHILE

// we will not process the copy if the destination is too small.
IF DestinationSize <> requiredDestinationSize THEN
	RETURN;
END_IF

currentPointer := DestinationAddress;
currentNode := First;

WHILE currentNode <> 0 DO
	currentNode.TryGetTo(currentPointer,currentNode.DataSize);
	currentPointer := currentPointer + currentNode.DataSize;
	currentNode := currentNode.Next;
END_WHILE
END_METHOD

METHOD PUBLIC TryRemoveItem : BOOL
VAR_INPUT
	Item : ANY;
END_VAR
VAR
	foundNode : I_LinkedListNode;
END_VAR
foundNode := FindFirstNodeWithValue(Item);

IF foundNode = 0 THEN
	RETURN;
END_IF

RemoveNode(foundNode);
EmitChangedEvent();

TryRemoveItem := TRUE;
END_METHOD

END_FUNCTION_BLOCK

// mobject-collections/Interfaces/Collections/Nodes/I_ListNode
INTERFACE I_ListNode EXTENDS I_CollectionNode;

END_INTERFACE

// mobject-collections/Interfaces/Collections/I_List
INTERFACE I_List EXTENDS I_Collection

PROPERTY PUBLIC Capacity : DINT
GET
END_GET
END_PROPERTY

METHOD PUBLIC GetIndexOf : DINT
VAR_INPUT
	Item : ANY;
END_VAR
END_METHOD

METHOD PUBLIC TrimExcess
END_METHOD

METHOD PUBLIC TryGetByIndex : BOOL
VAR_INPUT
	Index : DINT;
	Destination : ANY;
END_VAR
END_METHOD

METHOD PUBLIC TryGetToByIndex : BOOL
VAR_INPUT
	Index : DINT;
	DestinationAddress : PVOID;
	DestinationSize : UDINT;
END_VAR
END_METHOD

METHOD TryInsert : BOOL
VAR_INPUT
	Index : DINT;
	Item : ANY;
END_VAR
END_METHOD

METHOD TryRemoveAt : BOOL
VAR_INPUT
	Index : DINT;
END_VAR
END_METHOD

END_INTERFACE

// mobject-collections/Interfaces/Collections/I_Queue
INTERFACE I_Queue EXTENDS I_Collection

METHOD PUBLIC Enqueue
VAR_INPUT
	Item : ANY;
END_VAR
END_METHOD

METHOD PUBLIC TryDequeue : BOOL;
VAR_INPUT
	Destination : ANY;
END_VAR
END_METHOD

METHOD PUBLIC TryPeek : BOOL;
VAR_INPUT
	Destination : ANY;
END_VAR
END_METHOD

END_INTERFACE

// mobject-collections/Interfaces/Collections/I_Stack
INTERFACE I_Stack EXTENDS I_Collection

METHOD PUBLIC Push
VAR_INPUT
	Item : ANY;
END_VAR
END_METHOD

METHOD PUBLIC TryPeek : BOOL;
VAR_INPUT
	Destination : ANY;
END_VAR
END_METHOD

METHOD PUBLIC TryPop : BOOL;
VAR_INPUT
	Destination : ANY;
END_VAR
END_METHOD

END_INTERFACE

// mobject-collections/OrderedDictionary/OrderedDictionary
{attribute 'linkalways'} 
{attribute 'no_explicit_call' := 'This FB is a CLASS and must be accessed using methods or properties'}
{attribute 'enable_dynamic_creation'}
FUNCTION_BLOCK OrderedDictionary EXTENDS Disposable IMPLEMENTS I_Dictionary
VAR
	eventEmitter : EventEmitter;
	rootNode : I_OrderedDictionaryTreeNode;
	head : I_OrderedDictionaryTreeNode;
	tail : I_OrderedDictionaryTreeNode;
END_VAR

METHOD FB_exit : BOOL
VAR_INPUT
	bInCopyCode : BOOL; // if TRUE, the exit method is called for exiting an instance that is copied afterwards (online change).
END_VAR
VAR
END_VAR
IF bInCopyCode THEN
    RETURN;
END_IF

Clear();
EmitDisposedEvent();
END_METHOD

METHOD PRIVATE AddKeysInOrderToCollection
VAR_INPUT
	Collection : I_Collection;
END_VAR
VAR
	currentNode : I_OrderedDictionaryTreeNode;
	key : T_MAXSTRING;
END_VAR
IF head = 0 THEN
	RETURN;
END_IF

currentNode := head;

REPEAT
    key := currentNode.Key;
	Collection.AddItem(key);
	currentNode := currentNode.Next;
UNTIL
    currentNode = 0
END_REPEAT;
END_METHOD

METHOD PRIVATE AddNodesInOrderToCollection
VAR_INPUT
	Collection : I_Collection;
END_VAR
VAR
	currentNode : I_OrderedDictionaryTreeNode;
	key : T_MAXSTRING;
END_VAR
IF head = 0 THEN
	RETURN;
END_IF

currentNode := head;

REPEAT
	Collection.AddItem(currentNode);
	currentNode := currentNode.Next;
UNTIL
    currentNode = 0
END_REPEAT;
END_METHOD

METHOD PRIVATE AddNodeToEnd
VAR_INPUT
	Node : I_OrderedDictionaryTreeNode;
END_VAR
VAR
	originalTailNode : I_OrderedDictionaryTreeNode;
END_VAR
//LogMsg_I_OrderedDictionaryTreeNode('OrderedDictionary', 'AddNodeToEnd: Called with', Node);

IF head = 0 THEN
	head := Node;
	tail := Node;
	Node.Previous := 0;
	Node.Next := 0;
//	LogMsg('OrderedDictionary', 'AddNodeToEnd: Return, head = 0');
//	LogMsg_I_OrderedDictionaryTreeNode('OrderedDictionary', 'AddNodeToEnd: Head is', head);
//	LogMsg_I_OrderedDictionaryTreeNode('OrderedDictionary', 'AddNodeToEnd: Tail is', tail);
	RETURN;
END_IF

//LogMsg_I_OrderedDictionaryTreeNode('OrderedDictionary', 'AddNodeToEnd: Original Tail was', tail);
originalTailNode := tail;
tail := Node;
//LogMsg_I_OrderedDictionaryTreeNode('OrderedDictionary', 'AddNodeToEnd: Tail is now', tail);

originalTailNode.Next := node;
//LogMsg_I_OrderedDictionaryTreeNode('OrderedDictionary', 'AddNodeToEnd: Original Tail next is', originalTailNode.Next);
tail.Previous := originalTailNode;
tail.Next := 0;
//LogMsg_I_OrderedDictionaryTreeNode('OrderedDictionary', 'AddNodeToEnd: Tail previous is now', tail.Previous);

//LogMsg('OrderedDictionary', 'AddNodeToEnd: Return');
END_METHOD

METHOD PRIVATE Balance : I_OrderedDictionaryTreeNode
VAR_INPUT
	Node : I_OrderedDictionaryTreeNode;
END_VAR
VAR
	balanceFactor : DINT;
END_VAR
balanceFactor := THIS^.GetBalanceFactor(Node);

IF (balanceFactor > 1) THEN
	IF THIS^.GetBalanceFactor(Node.Left) < 0 THEN
		Node.Left := THIS^.LeftRotate(Node.Left);
	END_IF
	Node := RightRotate(Node);
ELSIF (balanceFactor < -1) THEN
	IF THIS^.GetBalanceFactor(Node.Right) > 0 THEN
		Node.Right := RightRotate(Node.Right);
	END_IF
	Node := LeftRotate(Node);
END_IF

Balance := Node;

//LogMsg('OrderedDictionary', ': Called');
//LogMsg_I_OrderedDictionaryTreeNode('OrderedDictionary', ': RootNode is now', rootNode);
//LogMsg('OrderedDictionary', ': Return');
END_METHOD

METHOD PRIVATE EmitChangedEvent
VAR
	dictionaryChangedEvent : KeyValueCollectionChangedEvent(Target := THIS^);
END_VAR
eventEmitter.Emit('OnChanged', dictionaryChangedEvent);
END_METHOD

METHOD PRIVATE EmitDisposedEvent
VAR
	dictionaryDisposedEvent : KeyValueCollectionDisposedEvent(Target := THIS^);
END_VAR
eventEmitter.Emit('OnDisposed', dictionaryDisposedEvent);
END_METHOD

METHOD PRIVATE FindMinimum : I_OrderedDictionaryTreeNode
VAR_INPUT
	Node : I_OrderedDictionaryTreeNode;
END_VAR
VAR
	nextNode : I_OrderedDictionaryTreeNode;
END_VAR
nextNode := Node;

WHILE (nextNode.left <> 0) DO
      nextNode := nextNode.left;
END_WHILE;

FindMinimum := nextNode;
END_METHOD

METHOD PRIVATE GetBalanceFactor : DINT
VAR_INPUT
	Node : I_OrderedDictionaryTreeNode;
END_VAR
IF (Node = 0) THEN
	GetBalanceFactor := 0;
	RETURN;
END_IF

GetBalanceFactor := THIS^.GetHeight(node.left) - THIS^.GetHeight(node.right);
END_METHOD

METHOD PRIVATE GetHeight : DINT
VAR_INPUT
	Node : I_OrderedDictionaryTreeNode;
END_VAR
IF Node = 0 THEN
	GetHeight := -1;
	RETURN;
END_IF

GetHeight := Node.Height;
END_METHOD

METHOD PRIVATE LeftRotate : I_OrderedDictionaryTreeNode
VAR_INPUT
	X : I_OrderedDictionaryTreeNode;
END_VAR
VAR
	y : I_OrderedDictionaryTreeNode;
	t2 : I_OrderedDictionaryTreeNode;
END_VAR
y := X.right;
t2 := y.left;
y.left := X;
X.right := t2;
THIS^.UpdateHeight(X);
THIS^.UpdateHeight(y);
LeftRotate := y;
END_METHOD

METHOD PRIVATE RecursiveCountNodes
VAR_INPUT
	Node : I_OrderedDictionaryTreeNode;
	Count : REFERENCE TO DINT;
END_VAR
IF Node = 0 THEN
	RETURN;
END_IF

Count := Count + 1;

THIS^.RecursiveCountNodes(Node.Left,Count);
THIS^.RecursiveCountNodes(Node.Right,Count);
END_METHOD

METHOD PRIVATE RecursiveDelete : I_OrderedDictionaryTreeNode
VAR_INPUT
	Key : T_MAXSTRING;
	Node : I_OrderedDictionaryTreeNode;
END_VAR
VAR
	newNode : I_OrderedDictionaryTreeNode; 
	minValueNode : I_OrderedDictionaryTreeNode;
	minValueNodeParent : I_OrderedDictionaryTreeNode;
	balanceFactor : DINT;
END_VAR
IF (Node = 0) THEN
    RETURN;
END_IF

IF (Key < Node.Key) THEN
    Node.left := THIS^.RecursiveDelete(Key, Node.left);
ELSIF (Key > Node.Key) THEN
    Node.right := THIS^.RecursiveDelete(Key, Node.right);
ELSE
    IF (Node.Left = 0) OR (Node.Right = 0) THEN
        IF (Node.Left = 0) THEN
            newNode := Node.Right;
        ELSE
            newNode := Node.Left;
        END_IF
		RemoveNodeFromLinkedList(Node);
        Node.Dispose();
        THIS^.updateHeight(newNode);
        RecursiveDelete := THIS^.Balance(newNode);
        RETURN;
    ELSE
		RemoveNodeFromLinkedList(Node);
		minValueNode := FindMinimum(Node.Right);
		ReplaceNodeInLinkedList(minValueNode, Node);
        Node.Right := THIS^.RecursiveDelete(minValueNode.Key, Node.Right);	
    END_IF
END_IF

THIS^.updateHeight(Node);
RecursiveDelete := THIS^.Balance(Node);
END_METHOD

METHOD PRIVATE RecursiveFind : I_OrderedDictionaryTreeNode
VAR_INPUT
	Key : T_MAXSTRING;
	Node : I_OrderedDictionaryTreeNode;
END_VAR
IF (Node = 0) THEN
	RETURN;
END_IF

IF (Key < Node.key) THEN
  RecursiveFind := THIS^.RecursiveFind(key, Node.left);
  RETURN;
ELSIF (key > Node.key) THEN
  RecursiveFind := THIS^.RecursiveFind(key, Node.right);
  RETURN;
ELSE 
  RecursiveFind := Node;
  RETURN;
END_IF
END_METHOD

METHOD PRIVATE RecursiveInsert : I_OrderedDictionaryTreeNode
VAR_INPUT
	Key : T_MAXSTRING;
	Value : ANY;
	Node : I_OrderedDictionaryTreeNode;
END_VAR
VAR
	pAVLTreeNode : POINTER TO OrderedDictionaryTreeNode;
	balanceFactor : DINT;
END_VAR
IF (Node = 0) THEN
	pAVLTreeNode := __NEW(OrderedDictionaryTreeNode(NodeKey := Key, NodeSource := Value));
	AddNodeToEnd(pAVLTreeNode^);
	RecursiveInsert := pAVLTreeNode^;
	RETURN;
END_IF

IF (Key < Node.Key) THEN
	Node.left := THIS^.RecursiveInsert(Key, Value, Node.left);
ELSIF (Key > Node.Key) THEN
	Node.right := THIS^.RecursiveInsert(Key, Value, Node.right);
ELSE
	Node.Reinitialize(Key,Value);
	RecursiveInsert := Node;
END_IF

THIS^.updateHeight(node);

balanceFactor := THIS^.GetBalanceFactor(Node);
Node := balance(Node);
RecursiveInsert := Node;
END_METHOD

METHOD PRIVATE RemoveNodeFromLinkedList
VAR_INPUT
	Node : I_OrderedDictionaryTreeNode;
END_VAR
VAR
	nodeBefore : I_OrderedDictionaryTreeNode; 
	nodeAfter : I_OrderedDictionaryTreeNode;
END_VAR
// if the node is the head and has no further nodes following it, then it must
// be the only node in the collection.  As such, set head, tail as 0.
IF Node = head AND Node = tail THEN
	head := 0;
	tail := 0;
	Node.Previous := 0;
	Node.Next := 0;
	RETURN;
END_IF

// if the node is at the start of more than one node, then
// make the next in line the head, and remove it's knowlege of
// the node being removed.
IF Node = head THEN
	Node.Next.Previous := 0;
	head := Node.Next;
	Node.Previous := 0;
	Node.Next := 0;
	RETURN;
END_IF

// if the node is at the end of more than one node, then
// make the previous in line the tail, and remove it's knowlege of
// the node being removed.
IF Node = tail THEN
	Node.Previous.Next := 0;
	tail := Node.Previous;
	Node.Previous := 0;
	Node.Next := 0;
	RETURN;
END_IF

// we need to perform this check as replaced nodes may not be head or tail
// but will have had the previous and next removed. Therefore only true deletes
// will have these set.
IF Node.Previous <> 0 AND Node.Next <> 0 THEN
	nodeBefore := Node.Previous;
	nodeAfter := Node.Next;	
	nodeBefore.Next := nodeAfter;
	nodeAfter.Previous := nodeBefore;
	Node.Next := 0;
	Node.Previous := 0;
END_IF
END_METHOD

METHOD PRIVATE ReplaceNodeInLinkedList
VAR_INPUT
	OldNode : I_OrderedDictionaryTreeNode;
	NewNode : I_OrderedDictionaryTreeNode;
END_VAR
// copy everything from the old node to the new node.
NewNode.DeepCopy(OldNode);

// if the node has a previous link, then that previous node will need to know that this
// ToNode is now its correct next as it will still be pointing to the old node.
IF OldNode.Previous <> 0 THEN
	OldNode.Previous.Next := NewNode;
END_IF
OldNode.Previous := 0;

// if the node has a next link, then that next node will need to know that this
// ToNode is now its correct next as it will still be pointing to the old node.
IF OldNode.Next <> 0 THEN
	OldNode.Next.Previous := NewNode;
END_IF
OldNode.Next := 0;

// if the head pointer was pointing at the old node then replace with new node.
if head = OldNode then
	head := NewNode;
END_IF

// if the tail pointer was pointing at the old node then replace with new node.
if tail = OldNode then
	tail := NewNode;
END_IF
END_METHOD

METHOD PRIVATE RightRotate : I_OrderedDictionaryTreeNode
VAR_INPUT
	Y : I_OrderedDictionaryTreeNode;
END_VAR
VAR
	x : I_OrderedDictionaryTreeNode;
	t2 : I_OrderedDictionaryTreeNode;
END_VAR
x := Y.left;
t2 := x.right;
x.right := Y;
Y.left := t2;
THIS^.UpdateHeight(Y);
THIS^.UpdateHeight(x);
RightRotate := x;
END_METHOD

METHOD PRIVATE UpdateHeight
VAR_INPUT
	Node : I_OrderedDictionaryTreeNode;
END_VAR
IF (Node = 0) THEN
	RETURN;
END_IF

Node.height := 1 + MAX(THIS^.GetHeight(Node.left), THIS^.GetHeight(Node.right));
END_METHOD

METHOD PUBLIC AddOrUpdate
VAR_INPUT
	Key : T_MAXSTRING;
	Value : ANY;
END_VAR
rootNode := THIS^.RecursiveInsert(Key, Value, rootNode);
EmitChangedEvent();
END_METHOD

METHOD PUBLIC Clear
VAR_INPUT
END_VAR
VAR
	currentNode : I_OrderedDictionaryTreeNode;
	nextNode : I_OrderedDictionaryTreeNode;
END_VAR
IF head = 0 THEN
	RETURN;
END_IF

currentNode := head;

WHILE currentNode <> 0 DO
	nextNode := currentNode.Next;
	currentNode.Dispose();
	currentNode := nextNode;
END_WHILE

head := 0;
tail := 0;
rootNode := 0;
EmitChangedEvent();
END_METHOD

METHOD PUBLIC ContainsKey : BOOL
VAR_INPUT
	Key : T_MAXSTRING;
END_VAR
VAR
	foundNode : I_OrderedDictionaryTreeNode;
END_VAR
foundNode := THIS^.RecursiveFind(Key, rootNode);

IF foundNode = 0 THEN
	RETURN;
END_IF

ContainsKey := TRUE;
END_METHOD

PROPERTY PUBLIC Count : DINT
GET
VAR
	NodeCount : DINT;
END_VAR
RecursiveCountNodes(rootNode, NodeCount);
Count := NodeCount;
END_GET
END_PROPERTY

METHOD GetEnumerator : I_ForwardEnumerator
VAR
	pNodeCollection : POINTER TO LinkedList;
	pEnumerator : POINTER TO OrderedDictionaryForwardEnumerator;
END_VAR
pNodeCollection := __NEW(LinkedList);
THIS^.AddNodesInOrderToCollection(pNodeCollection^);

pEnumerator := __NEW(OrderedDictionaryForwardEnumerator(Parent := THIS^, Nodes := pNodeCollection^));
GetEnumerator := pEnumerator^;
END_METHOD

METHOD PUBLIC GetKeys : I_Collection
VAR
	pLinkedList : POINTER TO LinkedList;
END_VAR
pLinkedList := __NEW(LinkedList);
THIS^.AddKeysInOrderToCollection(pLinkedList^);
GetKeys := pLinkedList^;
END_METHOD

METHOD GetKeyValueEnumerator : I_KeyValueForwardEnumerator
VAR
	pNodeCollection : POINTER TO LinkedList;
	pEnumerator : POINTER TO OrderedDictionaryForwardEnumerator;
END_VAR
pNodeCollection := __NEW(LinkedList);
THIS^.AddNodesInOrderToCollection(pNodeCollection^);

pEnumerator := __NEW(OrderedDictionaryForwardEnumerator(Parent := THIS^, Nodes := pNodeCollection^));
GetKeyValueEnumerator := pEnumerator^;
END_METHOD

PROPERTY IsEmpty : BOOL
GET
IsEmpty := rootNode = 0;
END_GET
END_PROPERTY

METHOD PUBLIC OffEvent
VAR_INPUT
	EventName : T_MaxString;
	EventHandler : I_EventHandler;
END_VAR
eventEmitter.OffEvent(EventName, EventHandler);
END_METHOD

METHOD PUBLIC OnceEvent
VAR_INPUT
	EventName : T_MaxString;
	EventHandler : I_EventHandler;
END_VAR
eventEmitter.OnceEvent(EventName, EventHandler);
END_METHOD

METHOD PUBLIC OnEvent
VAR_INPUT
	EventName : T_MaxString;
	EventHandler : I_EventHandler;
END_VAR
eventEmitter.OnEvent(EventName, EventHandler);
END_METHOD

METHOD PUBLIC Remove
VAR_INPUT
	Key : T_MAXSTRING;
END_VAR
rootNode := THIS^.RecursiveDelete(Key, rootNode);
EmitChangedEvent();
END_METHOD

METHOD PUBLIC TryAdd : BOOL
VAR_INPUT
	Key : T_MAXSTRING;
	Value : ANY;
END_VAR
IF ContainsKey(Key) THEN
	RETURN;
END_IF
	  
THIS^.AddOrUpdate(Key, Value);
TryAdd := TRUE;
END_METHOD

METHOD PUBLIC TryGetValue : BOOL
VAR_INPUT
	Key : T_MAXSTRING;
	Destination	: ANY;
END_VAR
TryGetValue := TryGetValueTo(Key, Destination.pValue, DINT_TO_UDINT(Destination.diSize));
END_METHOD

METHOD PUBLIC TryGetValueTo : BOOL
VAR_INPUT
	Key : T_MAXSTRING;
	DestinationAddress : PVOID;
	DestinationSize : UDINT;
END_VAR
VAR
	foundNode : I_OrderedDictionaryTreeNode;
END_VAR
foundNode := THIS^.RecursiveFind(Key, rootNode);

IF foundNode = 0 THEN
	RETURN;
END_IF

TryGetValueTo := foundNode.TryGetTo(DestinationAddress, DestinationSize);
END_METHOD

END_FUNCTION_BLOCK

// mobject-collections/Queue/Queue
{attribute 'linkalways'} 
{attribute 'no_explicit_call' := 'This FB is a CLASS and must be accessed using methods or properties'}
{attribute 'enable_dynamic_creation'}
FUNCTION_BLOCK Queue EXTENDS Disposable IMPLEMENTS I_Queue
VAR
	linkedList : LinkedList;
	eventEmitter : EventEmitter;
END_VAR

METHOD FB_exit : BOOL
VAR_INPUT
	bInCopyCode : BOOL; // if TRUE, the exit method is called for exiting an instance that is copied afterwards (online change).
END_VAR
IF bInCopyCode THEN
	RETURN;
END_IF

Clear();
EmitDisposedEvent();
END_METHOD

METHOD PRIVATE EmitChangedEvent
VAR
	pCollectionChangedEvent : POINTER TO CollectionChangedEvent;
END_VAR
pCollectionChangedEvent := __NEW(CollectionChangedEvent(Target := THIS^));
eventEmitter.Emit('OnChanged', pCollectionChangedEvent^);
pCollectionChangedEvent^.Dispose();
END_METHOD

METHOD PRIVATE EmitDisposedEvent
VAR
	pCollectionDisposedEvent : POINTER TO CollectionDisposedEvent;
END_VAR
pCollectionDisposedEvent := __NEW(CollectionDisposedEvent(Target := THIS^));
eventEmitter.Emit('OnDisposed', pCollectionDisposedEvent^);
pCollectionDisposedEvent^.Dispose();
END_METHOD

METHOD PUBLIC AddItem
VAR_INPUT
	Item : ANY;
END_VAR
Enqueue(Item);
END_METHOD

METHOD PUBLIC Clear
linkedList.Clear();
EmitChangedEvent();
END_METHOD

METHOD PUBLIC Contains : BOOL;
VAR_INPUT
	Item : ANY;
END_VAR
VAR
	found : I_LinkedListNode;
END_VAR
found := linkedList.Find(Item);
Contains := found <> 0;
END_METHOD

PROPERTY PUBLIC Count : DINT
GET
Count := linkedList.Count;
END_GET
END_PROPERTY

METHOD PUBLIC Enqueue
VAR_INPUT
	Item : ANY;
END_VAR
linkedList.AddLast(Item);
EmitChangedEvent();
END_METHOD

METHOD PUBLIC GetEnumerator : I_ForwardEnumerator
GetEnumerator := linkedList.GetEnumerator();
END_METHOD

PROPERTY IsEmpty : BOOL
GET
IsEmpty := linkedList.IsEmpty;
END_GET
END_PROPERTY

METHOD PUBLIC OffEvent
VAR_INPUT
	EventName : T_MaxString;
	EventHandler : I_EventHandler;
END_VAR
eventEmitter.OffEvent(EventName, EventHandler);
END_METHOD

METHOD PUBLIC OnceEvent
VAR_INPUT
	EventName : T_MaxString;
	EventHandler : I_EventHandler;
END_VAR
eventEmitter.OnceEvent(EventName, EventHandler);
END_METHOD

METHOD PUBLIC OnEvent
VAR_INPUT
	EventName : T_MaxString;
	EventHandler : I_EventHandler;
END_VAR
eventEmitter.OnEvent(EventName, EventHandler);
END_METHOD

METHOD PUBLIC TryCopyTo : BOOL
VAR_INPUT
	Destination : ANY;
END_VAR
TryCopyTo := linkedList.TryCopyTo(Destination);
END_METHOD

METHOD PUBLIC TryCopyToLocation : BOOL
VAR_INPUT
	DestinationAddress : PVOID;
	DestinationSize : UDINT;
END_VAR
TryCopyToLocation := linkedList.TryCopyToLocation(DestinationAddress, DestinationSize);
END_METHOD

METHOD PUBLIC TryDequeue : BOOL;
VAR_INPUT
	Destination : ANY;
END_VAR
VAR
	first : I_LinkedListNode;
	dequeued : BOOL;
END_VAR
first := linkedList.First;

IF first = 0 THEN
	RETURN;
END_IF

dequeued := linkedList.First.TryGet(Destination);

IF NOT dequeued THEN
	RETURN;
END_IF

linkedList.RemoveFirst();
EmitChangedEvent();
TryDequeue := TRUE;
END_METHOD

METHOD PUBLIC TryPeek : BOOL;
VAR_INPUT
	Destination : ANY;
END_VAR
VAR
	first : I_LinkedListNode;
END_VAR
first := linkedList.First;

IF first = 0 THEN
	RETURN;
END_IF

TryPeek := first.TryGet(Destination);
END_METHOD

METHOD PUBLIC TryRemoveItem : BOOL
VAR_INPUT
	Item : ANY;
END_VAR
TryRemoveItem := linkedList.TryRemoveItem(Item);
EmitChangedEvent();
END_METHOD

END_FUNCTION_BLOCK

// mobject-collections/Stack/Stack
{attribute 'linkalways'} 
{attribute 'no_explicit_call' := 'This FB is a CLASS and must be accessed using methods or properties'}
{attribute 'enable_dynamic_creation'}
FUNCTION_BLOCK Stack EXTENDS Disposable IMPLEMENTS I_Stack
VAR
	linkedList : LinkedList;
	eventEmitter : EventEmitter;
END_VAR

METHOD FB_exit : BOOL
VAR_INPUT
	bInCopyCode : BOOL; // if TRUE, the exit method is called for exiting an instance that is copied afterwards (online change).
END_VAR
IF bInCopyCode THEN
	RETURN;
END_IF

Clear();
EmitDisposedEvent();
END_METHOD

METHOD PRIVATE EmitChangedEvent
VAR
	pCollectionChangedEvent : POINTER TO CollectionChangedEvent;
END_VAR
pCollectionChangedEvent := __NEW(CollectionChangedEvent(Target := THIS^));
eventEmitter.Emit('OnChanged', pCollectionChangedEvent^);
pCollectionChangedEvent^.Dispose();
END_METHOD

METHOD PRIVATE EmitDisposedEvent
VAR
	pCollectionDisposedEvent : POINTER TO CollectionDisposedEvent;
END_VAR
pCollectionDisposedEvent := __NEW(CollectionDisposedEvent(Target := THIS^));
eventEmitter.Emit('OnDisposed', pCollectionDisposedEvent^);
pCollectionDisposedEvent^.Dispose();
END_METHOD

METHOD PUBLIC AddItem
VAR_INPUT
	Item : ANY;
END_VAR
Push(Item);
END_METHOD

METHOD PUBLIC Clear
linkedList.Clear();
EmitChangedEvent();
END_METHOD

METHOD PUBLIC Contains : BOOL;
VAR_INPUT
	Item : ANY;
END_VAR
VAR
	found : I_LinkedListNode;
END_VAR
found := linkedList.Find(Item);
Contains := found <> 0;
END_METHOD

PROPERTY PUBLIC Count : DINT
GET
Count := linkedList.Count;
END_GET
END_PROPERTY

METHOD PUBLIC GetEnumerator : I_ForwardEnumerator
GetEnumerator := linkedList.GetEnumerator();
END_METHOD

PROPERTY IsEmpty : BOOL
GET
IsEmpty := linkedList.IsEmpty;
END_GET
END_PROPERTY

METHOD PUBLIC OffEvent
VAR_INPUT
	EventName : T_MaxString;
	EventHandler : I_EventHandler;
END_VAR
eventEmitter.OffEvent(EventName, EventHandler);
END_METHOD

METHOD PUBLIC OnceEvent
VAR_INPUT
	EventName : T_MaxString;
	EventHandler : I_EventHandler;
END_VAR
eventEmitter.OnceEvent(EventName, EventHandler);
END_METHOD

METHOD PUBLIC OnEvent
VAR_INPUT
	EventName : T_MaxString;
	EventHandler : I_EventHandler;
END_VAR
eventEmitter.OnEvent(EventName, EventHandler);
END_METHOD

METHOD PUBLIC Push
VAR_INPUT
	Item : ANY;
END_VAR
linkedList.AddFirst(Item);
EmitChangedEvent();
END_METHOD

METHOD PUBLIC TryCopyTo : BOOL
VAR_INPUT
	Destination : ANY;
END_VAR
TryCopyTo := linkedList.TryCopyTo(Destination);
END_METHOD

METHOD PUBLIC TryCopyToLocation : BOOL
VAR_INPUT
	DestinationAddress : PVOID;
	DestinationSize : UDINT;
END_VAR
TryCopyToLocation := linkedList.TryCopyToLocation(DestinationAddress, DestinationSize);
END_METHOD

METHOD PUBLIC TryPeek : BOOL;
VAR_INPUT
	Destination : ANY;
END_VAR
VAR
	first : I_LinkedListNode;
END_VAR
first := linkedList.First;

IF first = 0 THEN
	RETURN;
END_IF

TryPeek := first.TryGet(Destination);
END_METHOD

METHOD PUBLIC TryPop : BOOL;
VAR_INPUT
	Destination : ANY;
END_VAR
VAR
	first : I_LinkedListNode;
	popped : BOOL;
END_VAR
first := linkedList.First;

IF first = 0 THEN
	RETURN;
END_IF

popped := linkedList.First.TryGet(Destination);

IF NOT popped THEN
	RETURN;
END_IF

linkedList.RemoveFirst();
EmitChangedEvent();
TryPop := TRUE;
END_METHOD

METHOD PUBLIC TryRemoveItem : BOOL
VAR_INPUT
	Item : ANY;
END_VAR
TryRemoveItem := linkedList.TryRemoveItem(Item);
EmitChangedEvent();
END_METHOD

END_FUNCTION_BLOCK

// mobject-commands/_Internal/AsyncCommandStateMachine/AsyncCommandStateMachine
{attribute 'linkalways'} 
{attribute 'no_explicit_call' := 'This FB is a CLASS and must be accessed using methods or properties'}
{attribute 'enable_dynamic_creation'}
FUNCTION_BLOCK AsyncCommandStateMachine IMPLEMENTS I_AsyncCommandStateControl
VAR
	state : (IDLE, INITIALIZING, EXECUTING, COMPLETING, COMPLETED, ABORTING, ABORTED, ERRORED);
	_errorId : UDINT;
END_VAR

METHOD PRIVATE StateComplete_Aborting
VAR_INPUT
END_VAR
state := ABORTED;
END_METHOD

METHOD PRIVATE StateComplete_Completing
VAR_INPUT
END_VAR
state := COMPLETED;
END_METHOD

METHOD PRIVATE StateComplete_Executing
VAR_INPUT
END_VAR
state := COMPLETING;
END_METHOD

METHOD PRIVATE StateComplete_Initializing
VAR_INPUT
END_VAR
state := EXECUTING;
END_METHOD

METHOD PUBLIC Abort
VAR_INPUT
END_VAR
CASE state OF
	IDLE : RETURN;
	ABORTING : RETURN;
	COMPLETED : RETURN;
	ABORTED : RETURN;
	ERRORED : RETURN;
END_CASE

state := ABORTING;
END_METHOD

METHOD PUBLIC Error
VAR_INPUT
	ErrorId : UDINT;
END_VAR
CASE state OF
	IDLE : RETURN;
	COMPLETED : RETURN;
	ABORTED : RETURN;
	ERRORED : RETURN;
END_CASE

_errorId := ErrorId;
state := ERRORED;
END_METHOD

{attribute 'monitoring' := 'call'}
PROPERTY PUBLIC ErrorId : UDINT
GET
ErrorID := _errorId;
END_GET
END_PROPERTY

METHOD PUBLIC Execute
VAR_INPUT
END_VAR
CASE state OF
	INITIALIZING : RETURN;
	EXECUTING : RETURN;
	COMPLETING : RETURN;
	ABORTING : RETURN;
END_CASE

_errorId := 0;
state := INITIALIZING;
END_METHOD

{attribute 'monitoring' := 'call'}
PROPERTY PUBLIC IsAborted : BOOL
GET
IsAborted := state = ABORTED;
END_GET
END_PROPERTY

{attribute 'monitoring' := 'call'}
PROPERTY PUBLIC IsAborting : BOOL
GET
IsAborting := state = ABORTING;
END_GET
END_PROPERTY

{attribute 'monitoring' := 'call'}
PROPERTY PUBLIC IsCompleted : BOOL
GET
IsCompleted := state = COMPLETED;
END_GET
END_PROPERTY

{attribute 'monitoring' := 'call'}
PROPERTY PUBLIC IsCompleting : BOOL
GET
IsCompleting := state = COMPLETING;
END_GET
END_PROPERTY

{attribute 'monitoring' := 'call'}
PROPERTY PUBLIC IsErrored : BOOL
GET
IsErrored := state = ERRORED;
END_GET
END_PROPERTY

{attribute 'monitoring' := 'call'}
PROPERTY PUBLIC IsExecuting : BOOL
GET
IsExecuting := state = EXECUTING;
END_GET
END_PROPERTY

{attribute 'monitoring' := 'call'}
PROPERTY PUBLIC IsIdle : BOOL
GET
IsIdle:= state = IDLE;
END_GET
END_PROPERTY

{attribute 'monitoring' := 'call'}
PROPERTY PUBLIC IsInitializing : BOOL
GET
IsInitializing := state = INITIALIZING;
END_GET
END_PROPERTY

METHOD PUBLIC Next
VAR_INPUT
END_VAR
CASE state OF
	IDLE : RETURN;
	INITIALIZING : StateComplete_Initializing();
	EXECUTING : StateComplete_Executing();
	COMPLETING : StateComplete_Completing();
	COMPLETED : RETURN;
	ABORTING : StateComplete_Aborting();
	ABORTED : RETURN;
	ERRORED : RETURN;
END_CASE
END_METHOD

END_FUNCTION_BLOCK

// mobject-commands/_Internal/AsyncCommandStateMachine/I_AsyncCommandStateControl
INTERFACE I_AsyncCommandStateControl

METHOD PUBLIC Error
VAR_INPUT
	ErrorId : UDINT;
END_VAR
END_METHOD

METHOD PUBLIC Next
VAR_INPUT
END_VAR
END_METHOD

END_INTERFACE

// mobject-errors/Errors/Error
{attribute 'linkalways'} 
{attribute 'no_explicit_call' := 'This FB is a CLASS and must be accessed using methods or properties'}
{attribute 'enable_dynamic_creation'}
FUNCTION_BLOCK ABSTRACT Error EXTENDS Disposable IMPLEMENTS I_Error
VAR
END_VAR

METHOD PROTECTED OnSerialize
VAR_INPUT
	Serializer : I_Serializer;
END_VAR
END_METHOD

METHOD PUBLIC Accept
VAR_INPUT
	Visitor : I_ErrorVisitor;
END_VAR
Visitor.VisitError(THIS^);
END_METHOD

PROPERTY PUBLIC ABSTRACT ErrorType : T_MAXSTRING
GET
END_GET
END_PROPERTY

METHOD PUBLIC IsSameAs : BOOL
VAR_INPUT
	Error : I_Error;
END_VAR
IF Error = 0 THEN
	RETURN;
END_IF

IF Error.ErrorType <> THIS^.ErrorType THEN
	RETURN;
END_IF

IsSameAs := TRUE;
END_METHOD

PROPERTY PUBLIC ABSTRACT Message : T_MAXSTRING
GET
END_GET
END_PROPERTY

METHOD PUBLIC SerializeWith
VAR_INPUT
	Serializer : I_Serializer;
END_VAR
Serializer.StartObject();
Serializer.AddKeyString('errorType',ErrorType);
Serializer.AddKeyString('message',Message);
OnSerialize(Serializer);
Serializer.EndObject();
END_METHOD

END_FUNCTION_BLOCK

// mobject-errors/Interfaces/I_Error
INTERFACE I_Error EXTENDS I_Serializable, I_Disposable

METHOD PUBLIC Accept
VAR_INPUT
	Visitor : I_ErrorVisitor;
END_VAR
END_METHOD

PROPERTY ErrorType : T_MAXSTRING
GET
END_GET
END_PROPERTY

METHOD PUBLIC IsSameAs : BOOL
VAR_INPUT
	Error : I_Error;
END_VAR
END_METHOD

PROPERTY Message : T_MAXSTRING
GET
END_GET
END_PROPERTY

END_INTERFACE

// mobject-serialization/Interfaces/I_Serializable
INTERFACE I_Serializable EXTENDS __SYSTEM.IQueryInterface

METHOD SerializeWith
VAR_INPUT
	Serializer : I_Serializer;
END_VAR
END_METHOD

END_INTERFACE

// mobject-serialization/Interfaces/I_Serializer
INTERFACE I_Serializer EXTENDS I_Disposable

METHOD PUBLIC AddBase64 : I_Serializer
VAR_INPUT
	pBytes : POINTER TO BYTE;
	nBytes : DINT;
END_VAR
END_METHOD

METHOD PUBLIC AddBool : I_Serializer
VAR_INPUT
	Value : BOOL;
END_VAR
END_METHOD

METHOD PUBLIC AddByte : I_Serializer
VAR_INPUT
	Value : BYTE;
END_VAR
END_METHOD

METHOD PUBLIC AddBytesAsHex : I_Serializer
VAR_INPUT
	pBytes : POINTER TO BYTE;
	nBytes : DINT;
END_VAR
END_METHOD

METHOD PUBLIC AddDateTime : I_Serializer
VAR_INPUT
	Value : DATE_AND_TIME;
END_VAR
END_METHOD

METHOD PUBLIC AddDcTime : I_Serializer
VAR_INPUT
	Value : DCTIME;
END_VAR
END_METHOD

METHOD PUBLIC AddDint : I_Serializer
VAR_INPUT
	Value : DINT;
END_VAR
END_METHOD

METHOD PUBLIC AddDword : I_Serializer
VAR_INPUT
	Value : DWORD;
END_VAR
END_METHOD

METHOD PUBLIC AddFileTime : I_Serializer
VAR_INPUT
	Value : FILETIME;
END_VAR
END_METHOD

METHOD PUBLIC AddInt : I_Serializer
VAR_INPUT
	Value : INT;
END_VAR
END_METHOD

METHOD PUBLIC AddKey : I_Serializer
VAR_INPUT
	Key : T_MAXSTRING;
END_VAR
END_METHOD

METHOD PUBLIC AddKeyBase64 : I_Serializer
VAR_INPUT
	Key : T_MAXSTRING;
	pBytes : POINTER TO BYTE;
	nBytes : DINT;
END_VAR
END_METHOD

METHOD PUBLIC AddKeyBool : I_Serializer
VAR_INPUT
	Key : T_MAXSTRING;
	Value : BOOL;
END_VAR
END_METHOD

METHOD PUBLIC AddKeyByte : I_Serializer
VAR_INPUT
	Key : T_MAXSTRING;
	Value : BYTE;
END_VAR
END_METHOD

METHOD PUBLIC AddKeyBytesAsHex : I_Serializer
VAR_INPUT
	Key : T_MAXSTRING;
	pBytes : POINTER TO BYTE;
	nBytes : DINT;
END_VAR
END_METHOD

METHOD PUBLIC AddKeyDateTime : I_Serializer
VAR_INPUT
	Key : T_MAXSTRING;
	Value : DATE_AND_TIME;
END_VAR
END_METHOD

METHOD PUBLIC AddKeyDcTime : I_Serializer
VAR_INPUT
	Key : T_MAXSTRING;
	Value : DCTIME;
END_VAR
END_METHOD

METHOD PUBLIC AddKeyDint : I_Serializer
VAR_INPUT
	Key : T_MAXSTRING;
	Value : DINT;
END_VAR
END_METHOD

METHOD PUBLIC AddKeyDword : I_Serializer
VAR_INPUT
	Key : T_MAXSTRING;
	Value : DWORD;
END_VAR
END_METHOD

METHOD PUBLIC AddKeyFileTime : I_Serializer
VAR_INPUT
	Key : T_MAXSTRING;
	Value : FILETIME;
END_VAR
END_METHOD

METHOD PUBLIC AddKeyInt : I_Serializer
VAR_INPUT
	Key : T_MAXSTRING;
	Value : INT;
END_VAR
END_METHOD

METHOD PUBLIC AddKeyLint : I_Serializer
VAR_INPUT
	Key : T_MAXSTRING;
	Value : LINT;
END_VAR
END_METHOD

METHOD PUBLIC AddKeyLreal : I_Serializer
VAR_INPUT
	Key : T_MAXSTRING;
	Value : LREAL;
END_VAR
END_METHOD

METHOD PUBLIC AddKeyLtime : I_Serializer
VAR_INPUT
	Key : T_MAXSTRING;
	Value : LTIME;
END_VAR
END_METHOD

METHOD PUBLIC AddKeyLword : I_Serializer
VAR_INPUT
	Key : T_MAXSTRING;
	Value : LWORD;
END_VAR
END_METHOD

METHOD PUBLIC AddKeyNull : I_Serializer
VAR_INPUT
	Key : T_MAXSTRING;
END_VAR
END_METHOD

METHOD PUBLIC AddKeyObject : I_Serializer
VAR_INPUT
	Key : T_MAXSTRING;
	Object : I_Serializable;
END_VAR
END_METHOD

METHOD PUBLIC AddKeyReal : I_Serializer
VAR_INPUT
	Key : T_MAXSTRING;
	Value : REAL;
END_VAR
END_METHOD

METHOD PUBLIC AddKeySint : I_Serializer
VAR_INPUT
	Key : T_MAXSTRING;
	Value : SINT;
END_VAR
END_METHOD

METHOD PUBLIC AddKeyString : I_Serializer
VAR_INPUT
	Key : T_MAXSTRING;
	Value : T_MAXSTRING;
END_VAR
END_METHOD

METHOD PUBLIC AddKeyStringByRef : I_Serializer
VAR_INPUT
	Key : T_MAXSTRING;
	Value : REFERENCE TO STRING;
END_VAR
END_METHOD

METHOD PUBLIC AddKeyTime : I_Serializer
VAR_INPUT
	Key : T_MAXSTRING;
	Value : TIME;
END_VAR
END_METHOD

METHOD PUBLIC AddKeyTod : I_Serializer
VAR_INPUT
	Key : T_MAXSTRING;
	Value : TOD;
END_VAR
END_METHOD

METHOD PUBLIC AddKeyUdint : I_Serializer
VAR_INPUT
	Key : T_MAXSTRING;
	Value : UDINT;
END_VAR
END_METHOD

METHOD PUBLIC AddKeyUint : I_Serializer
VAR_INPUT
	Key : T_MAXSTRING;
	Value : UINT;
END_VAR
END_METHOD

METHOD PUBLIC AddKeyUlint : I_Serializer
VAR_INPUT
	Key : T_MAXSTRING;
	Value : ULINT;
END_VAR
END_METHOD

METHOD PUBLIC AddKeyUsint : I_Serializer
VAR_INPUT
	Key : T_MAXSTRING;
	Value : USINT;
END_VAR
END_METHOD

METHOD PUBLIC AddKeyWord : I_Serializer
VAR_INPUT
	Key : T_MAXSTRING;
	Value : WORD;
END_VAR
END_METHOD

METHOD PUBLIC AddLint : I_Serializer
VAR_INPUT
	Value : LINT;
END_VAR
END_METHOD

METHOD PUBLIC AddLreal : I_Serializer
VAR_INPUT
	Value : LREAL;
END_VAR
END_METHOD

METHOD PUBLIC AddLtime : I_Serializer
VAR_INPUT
	Value : LTIME;
END_VAR
END_METHOD

METHOD PUBLIC AddLword : I_Serializer
VAR_INPUT
	Value : LWORD;
END_VAR
END_METHOD

METHOD PUBLIC AddNull : I_Serializer
VAR_INPUT
END_VAR
END_METHOD

METHOD PUBLIC AddObject
VAR_INPUT
	Object : I_Serializable;
END_VAR
END_METHOD

METHOD PUBLIC AddReal : I_Serializer
VAR_INPUT
	Value : REAL;
END_VAR
END_METHOD

METHOD PUBLIC AddSint : I_Serializer
VAR_INPUT
	Value : SINT;
END_VAR
END_METHOD

METHOD PUBLIC AddString : I_Serializer
VAR_INPUT
	Value : T_MAXSTRING;
END_VAR
END_METHOD

METHOD PUBLIC AddStringByRef : I_Serializer
VAR_INPUT
	Value : REFERENCE TO STRING;
END_VAR
END_METHOD

METHOD PUBLIC AddTime : I_Serializer
VAR_INPUT
	Value : TIME;
END_VAR
END_METHOD

METHOD PUBLIC AddTod : I_Serializer
VAR_INPUT
	Value : TOD;
END_VAR
END_METHOD

METHOD PUBLIC AddUdint : I_Serializer
VAR_INPUT
	Value : UDINT;
END_VAR
END_METHOD

METHOD PUBLIC AddUint : I_Serializer
VAR_INPUT
	Value : UINT;
END_VAR
END_METHOD

METHOD PUBLIC AddUlint : I_Serializer
VAR_INPUT
	Value : ULINT;
END_VAR
END_METHOD

METHOD PUBLIC AddUsint : I_Serializer
VAR_INPUT
	Value : USINT;
END_VAR
END_METHOD

METHOD PUBLIC AddWord : I_Serializer
VAR_INPUT
	Value : WORD;
END_VAR
END_METHOD

METHOD PUBLIC Clone : I_Serializer
END_METHOD

METHOD PUBLIC EndArray : I_Serializer
VAR_INPUT
END_VAR
END_METHOD

METHOD PUBLIC EndObject : I_Serializer
VAR_INPUT
END_VAR
END_METHOD

METHOD PUBLIC GetSerializedDataLength : UDINT
VAR_INPUT
END_VAR
END_METHOD

METHOD PUBLIC Reset
VAR_INPUT
END_VAR
END_METHOD

METHOD PUBLIC StartArray : I_Serializer
VAR_INPUT
END_VAR
END_METHOD

METHOD PUBLIC StartObject : I_Serializer
VAR_INPUT
END_VAR
END_METHOD

METHOD TryCopySerializedData : BOOL
VAR_INPUT
	DestinationAddress : PVOID;
	DestinationSize : UDINT;
END_VAR
END_METHOD

METHOD TryGetSerializedData : BOOL
VAR_INPUT
	DestinationAddress : PVOID;
	DestinationSize : UDINT;
END_VAR
END_METHOD

END_INTERFACE

// mobject-errors/Interfaces/I_ErrorVisitor
INTERFACE I_ErrorVisitor

METHOD VisitError
VAR_INPUT
	VisitingError : I_Error;
END_VAR
END_METHOD

END_INTERFACE

// mobject-commands/AsyncCommand/Interface/I_AsyncCommand
INTERFACE I_AsyncCommand extends I_Command

METHOD PUBLIC Abort
VAR_INPUT
END_VAR
END_METHOD

PROPERTY PUBLIC Busy : BOOL
GET
END_GET
END_PROPERTY

METHOD PUBLIC CyclicCall
VAR_INPUT
END_VAR
END_METHOD

PROPERTY PUBLIC Done : BOOL
GET
END_GET
END_PROPERTY

PROPERTY PUBLIC Error : BOOL
GET
END_GET
END_PROPERTY

PROPERTY PUBLIC ErrorId : UDINT
GET
END_GET
END_PROPERTY

END_INTERFACE

// mobject-commands/Command/Interface/I_Command
INTERFACE I_Command EXTENDS I_Disposable

METHOD Execute
VAR_INPUT
END_VAR
END_METHOD

END_INTERFACE

// mobject-commands/AsyncCommand/Runners/SingleAsyncCommandRunner
{attribute 'linkalways'} 
{attribute 'no_explicit_call' := 'This FB is a CLASS and must be accessed using methods or properties'}
{attribute 'enable_dynamic_creation'}
FUNCTION_BLOCK SingleAsyncCommandRunner
VAR
	currentCommand : I_AsyncCommand;
	replacementCommand : I_AsyncCommand;
END_VAR

PROPERTY PUBLIC Busy : BOOL
GET
IF currentCommand = 0 THEN
	RETURN;
END_IF

Busy := currentCommand.Busy;
END_GET
END_PROPERTY

METHOD PUBLIC CyclicCall
VAR_INPUT
END_VAR
IF currentCommand <> 0 AND_THEN currentCommand.Busy THEN
	currentCommand.CyclicCall();
	RETURN;
END_IF

IF replacementCommand <> 0 THEN
	currentCommand := replacementCommand;
	replacementCommand := 0;
	currentCommand.Execute();
END_IF
END_METHOD

PROPERTY Done : BOOL
GET
IF currentCommand = 0 THEN
	RETURN;
END_IF

Done := currentCommand.Done;
END_GET
END_PROPERTY

PROPERTY Error : BOOL
GET
IF currentCommand = 0 THEN
	RETURN;
END_IF

Error := currentCommand.Error;
END_GET
END_PROPERTY

PROPERTY PUBLIC ErrorId : UDINT
GET
IF currentCommand = 0 THEN
	RETURN;
END_IF

ErrorId := currentCommand.ErrorId;
END_GET
END_PROPERTY

METHOD ExecuteCommand
VAR_INPUT
	Command : I_AsyncCommand;
END_VAR
IF currentCommand = 0 THEN
	currentCommand := Command;
	currentCommand.Execute();
	RETURN;
END_IF

currentCommand.Abort();
replacementCommand := Command;
END_METHOD

END_FUNCTION_BLOCK

// mobject-commands/AsyncCommand/AsyncCommand
{attribute 'linkalways'} 
{attribute 'no_explicit_call' := 'This FB is a CLASS and must be accessed using methods or properties'}
{attribute 'enable_dynamic_creation'}
FUNCTION_BLOCK AsyncCommand EXTENDS Disposable IMPLEMENTS I_AsyncCommand
VAR
	stateMachine : AsyncCommandStateMachine;
END_VAR

METHOD PROTECTED OnAborted
VAR_INPUT
END_VAR
END_METHOD

METHOD PROTECTED OnAborting
VAR_INPUT
	StateControl : I_AsyncCommandStateControl;
END_VAR
// default behaviour is to go to next state
// you can override this method to implement your own completing control code.
// just call StateControl.Next() when your code is completed.  

StateControl.Next();
END_METHOD

METHOD PROTECTED OnCompleted : BOOL
VAR_INPUT
END_VAR
END_METHOD

METHOD PROTECTED OnCompleting
VAR_INPUT
	StateControl : I_AsyncCommandStateControl;
END_VAR
// default behaviour is to go to next state
// you can override this method to implement your own completing control code.
// just call StateControl.Next() when your code is completed.  

StateControl.Next();
END_METHOD

METHOD PROTECTED OnErrored
VAR_INPUT
END_VAR
END_METHOD

METHOD PROTECTED OnExecuting
VAR_INPUT
	StateControl : I_AsyncCommandStateControl;
END_VAR
// default behaviour is to go to next state
// you can override this method to implement your own executing control code.
// just call StateControl.Next() when your code is completed.  

StateControl.Next();
END_METHOD

METHOD PROTECTED OnIdle
VAR_INPUT
END_VAR
END_METHOD

METHOD PROTECTED OnInitializing
VAR_INPUT
	StateControl : I_AsyncCommandStateControl;
END_VAR
// default behaviour is to go to next state
// you can override this method to implement your own initializing control code.
// just call StateControl.Next() when your code is completed.  

StateControl.Next();
END_METHOD

METHOD PUBLIC Abort
VAR_INPUT
END_VAR
stateMachine.Abort();
END_METHOD

PROPERTY PUBLIC Busy : BOOL
GET
IF stateMachine.IsAborted THEN
	RETURN;
END_IF

IF stateMachine.IsCompleted THEN
	RETURN;
END_IF

IF stateMachine.IsErrored THEN
	RETURN;
END_IF

IF stateMachine.IsIdle THEN
	RETURN;
END_IF

Busy := TRUE;
END_GET
END_PROPERTY

METHOD PUBLIC CyclicCall
VAR_INPUT
END_VAR
IF stateMachine.IsIdle THEN
	OnIdle();
END_IF

IF stateMachine.IsInitializing THEN
	OnInitializing(stateMachine);
END_IF

IF stateMachine.IsExecuting THEN
	OnExecuting(stateMachine);
END_IF

IF stateMachine.IsCompleting THEN
	OnCompleting(stateMachine);
END_IF

IF stateMachine.IsCompleted THEN
	OnCompleted();
END_IF

IF stateMachine.IsAborting THEN
	OnAborting(stateMachine);
END_IF

IF stateMachine.IsAborted THEN
	OnAborted();
END_IF

IF stateMachine.IsErrored THEN
	OnErrored();
END_IF
END_METHOD

PROPERTY PUBLIC Done : BOOL
GET
Done := stateMachine.IsCompleted;
END_GET
END_PROPERTY

PROPERTY PUBLIC Error : BOOL
GET
Error := stateMachine.IsErrored;
END_GET
END_PROPERTY

PROPERTY PUBLIC ErrorId : UDINT
GET
ErrorId := stateMachine.ErrorId;
END_GET
END_PROPERTY

METHOD PUBLIC Execute
VAR_INPUT
END_VAR
stateMachine.Execute();
END_METHOD

END_FUNCTION_BLOCK

// mobject-converters/Converters/BOOL_TO_/TryConvert_BOOL_TO_BOOL
FUNCTION TryConvert_BOOL_TO_BOOL : BOOL
VAR_INPUT
	in : BOOL;
	out : REFERENCE TO BOOL;
END_VAR

out := in;
TryConvert_BOOL_TO_BOOL := TRUE;

END_FUNCTION

// mobject-converters/Converters/BOOL_TO_/TryConvert_BOOL_TO_BYTE
FUNCTION TryConvert_BOOL_TO_BYTE : BOOL
VAR_INPUT
	in : BOOL;
	out : REFERENCE TO BYTE;
END_VAR

out := BOOL_TO_BYTE(in);
TryConvert_BOOL_TO_BYTE := TRUE;

END_FUNCTION

// mobject-converters/Converters/BOOL_TO_/TryConvert_BOOL_TO_DATE
FUNCTION TryConvert_BOOL_TO_DATE : BOOL
VAR_INPUT
	in : BOOL;
	out : REFERENCE TO DATE;
END_VAR

out := BOOL_TO_DATE(in);
TryConvert_BOOL_TO_DATE := TRUE;

END_FUNCTION

// mobject-converters/Converters/BOOL_TO_/TryConvert_BOOL_TO_Destination
FUNCTION TryConvert_BOOL_TO_Destination : BOOL
VAR_INPUT
	in : BOOL;
	out : ANY;
END_VAR
VAR
	convertResult : BOOL := FALSE;
	convertAddress : PVOID;
	_BOOL : BOOL;
	_BYTE : BYTE;
	_WORD : WORD;
	_DWORD : DWORD;
	_LWORD : LWORD;
	_SINT : SINT;
	_INT : INT;
	_DINT : DINT;
	_LINT : LINT;
	_USINT : USINT;
	_UINT : UINT;
	_UDINT : UDINT;
	_ULINT : ULINT;
	_REAL : REAL;
	_LREAL : LREAL;
	_TIME : TIME;
	_TOD : TOD;
	_DATE : DATE;
	_DT : DT;
	_STRING : STRING;
END_VAR

CASE out.TypeClass OF
	__SYSTEM.TYPE_CLASS.TYPE_BOOL:
	
	convertResult := TryConvert_BOOL_TO_BOOL(in, _BOOL);
	IF convertResult THEN
		convertAddress := ADR(_BOOL);
	END_IF
	
	__SYSTEM.TYPE_CLASS.TYPE_BYTE:
	
	convertResult := TryConvert_BOOL_TO_BYTE(in, _BYTE);
	IF convertResult THEN
		convertAddress := ADR(_BYTE);
	END_IF
	
	__SYSTEM.TYPE_CLASS.TYPE_WORD:
	
	convertResult := TryConvert_BOOL_TO_WORD(in, _WORD);
	IF convertResult THEN
		convertAddress := ADR(_WORD);
	END_IF
	
	__SYSTEM.TYPE_CLASS.TYPE_DWORD:
	
	convertResult := TryConvert_BOOL_TO_DWORD(in, _DWORD);
	IF convertResult THEN
		convertAddress := ADR(_DWORD);
	END_IF
	
	__SYSTEM.TYPE_CLASS.TYPE_LWORD:
	
	convertResult := TryConvert_BOOL_TO_LWORD(in, _LWORD);
	IF convertResult THEN
		convertAddress := ADR(_LWORD);
	END_IF
	
	__SYSTEM.TYPE_CLASS.TYPE_SINT:
	
	convertResult := TryConvert_BOOL_TO_SINT(in, _SINT);
	IF convertResult THEN
		convertAddress := ADR(_SINT);
	END_IF
	
	__SYSTEM.TYPE_CLASS.TYPE_INT:
	
	convertResult := TryConvert_BOOL_TO_INT(in, _INT);
	IF convertResult THEN
		convertAddress := ADR(_INT);
	END_IF
	
	__SYSTEM.TYPE_CLASS.TYPE_DINT:
	
	convertResult := TryConvert_BOOL_TO_DINT(in, _DINT);
	IF convertResult THEN
		convertAddress := ADR(_DINT);
	END_IF
	
	__SYSTEM.TYPE_CLASS.TYPE_LINT:
	
	convertResult := TryConvert_BOOL_TO_LINT(in, _LINT);
	IF convertResult THEN
		convertAddress := ADR(_LINT);
	END_IF
	
	__SYSTEM.TYPE_CLASS.TYPE_USINT:
	
	convertResult := TryConvert_BOOL_TO_USINT(in, _USINT);
	IF convertResult THEN
		convertAddress := ADR(_USINT);
	END_IF
	
	__SYSTEM.TYPE_CLASS.TYPE_UINT:
	
	convertResult := TryConvert_BOOL_TO_UINT(in, _UINT);
	IF convertResult THEN
		convertAddress := ADR(_UINT);
	END_IF
	
	__SYSTEM.TYPE_CLASS.TYPE_UDINT:
	
	convertResult := TryConvert_BOOL_TO_UDINT(in, _UDINT);
	IF convertResult THEN
		convertAddress := ADR(_UDINT);
	END_IF
	
	__SYSTEM.TYPE_CLASS.TYPE_ULINT:
	
	convertResult := TryConvert_BOOL_TO_ULINT(in, _ULINT);
	IF convertResult THEN
		convertAddress := ADR(_ULINT);
	END_IF
	
	__SYSTEM.TYPE_CLASS.TYPE_REAL:
	
	convertResult := TryConvert_BOOL_TO_REAL(in, _REAL);
	IF convertResult THEN
		convertAddress := ADR(_REAL);
	END_IF
	
	__SYSTEM.TYPE_CLASS.TYPE_LREAL:
	
	convertResult := TryConvert_BOOL_TO_LREAL(in, _LREAL);
	IF convertResult THEN
		convertAddress := ADR(_LREAL);
	END_IF
	
	__SYSTEM.TYPE_CLASS.TYPE_TIME:
	
	convertResult := TryConvert_BOOL_TO_TIME(in, _TIME);
	IF convertResult THEN
		convertAddress := ADR(_TIME);
	END_IF
	
	__SYSTEM.TYPE_CLASS.TYPE_TIMEOFDAY:
	
	convertResult := TryConvert_BOOL_TO_TOD(in, _TOD);
	IF convertResult THEN
		convertAddress := ADR(_TOD);
	END_IF
	
	__SYSTEM.TYPE_CLASS.TYPE_DATE:
	
	convertResult := TryConvert_BOOL_TO_DATE(in, _DATE);
	IF convertResult THEN
		convertAddress := ADR(_DATE);
	END_IF
	
	__SYSTEM.TYPE_CLASS.TYPE_DATEANDTIME:
	
	convertResult := TryConvert_BOOL_TO_DT(in, _DT);
	IF convertResult THEN
		convertAddress := ADR(_DT);
	END_IF
	
	__SYSTEM.TYPE_CLASS.TYPE_STRING:
	
	convertResult := TryConvert_BOOL_TO_STRING(in, _STRING);
	IF convertResult THEN
		convertAddress := ADR(_STRING);
	END_IF
	
END_CASE

IF convertResult THEN
	memcpy(out.pValue,convertAddress,DINT_TO_UDINT(out.diSize));
END_IF

TryConvert_BOOL_TO_Destination := convertResult;

END_FUNCTION

// mobject-datatypes/Primitive/_BOOL
{attribute 'linkalways'} 
{attribute 'no_explicit_call' := 'This FB is a CLASS and must be accessed using methods or properties'}
{attribute 'enable_dynamic_creation'}
FUNCTION_BLOCK _BOOL EXTENDS DatatypeBase IMPLEMENTS I_BOOL
VAR
	localData : BOOL;
	activeData : REFERENCE TO BOOL REF= localData;
END_VAR

METHOD FB_init : BOOL
VAR_INPUT
	bInitRetains : BOOL; // if TRUE, the retain variables are initialized (warm start / cold start)
	bInCopyCode : BOOL;  // if TRUE, the instance afterwards gets moved into the copy code (online change)
	InitialValue : BOOL;
END_VAR
localData := InitialValue;
END_METHOD

PROPERTY PUBLIC Address : PVOID
GET
Address := ADR(activeData);
END_GET
END_PROPERTY

METHOD PUBLIC ClearReference
VAR_INPUT
END_VAR
activeData REF= localData;
END_METHOD

METHOD PUBLIC Clone : I_Datatype
VAR
    pClone : POINTER TO _BOOL;
END_VAR
pClone := __NEW(_BOOL(InitialValue := Value));
Clone := pClone^;
END_METHOD

METHOD PUBLIC MakeReferenceTo
VAR_INPUT
	ReferenceTarget : REFERENCE TO BOOL;
END_VAR
activeData REF= ReferenceTarget;
END_METHOD

METHOD PUBLIC SerializeWith
VAR_INPUT
	Serializer : I_Serializer;
END_VAR
Serializer.AddBool(activeData);
END_METHOD

PROPERTY PUBLIC Size : UDINT
GET
Size := SIZEOF(activeData);
END_GET
END_PROPERTY

METHOD PUBLIC TryConvertTo : BOOL
VAR_INPUT
	Destination : ANY;
END_VAR
TryConvertTo := TryConvert_BOOL_To_Destination(activeData, Destination);
END_METHOD

METHOD PUBLIC TryConvertTo_ : BOOL
VAR_INPUT
	Destination : I_Datatype;
END_VAR
VAR
	resultofBitConversion : BOOL;
	destinationAs_BIT : I_BIT;
	destinationAs_BOOL : I_BOOL;
	destinationAs_BYTE : I_BYTE;
	destinationAs_DINT : I_DINT;
	destinationAs_DT : I_DT;
	destinationAs_DWORD : I_DWORD;
	destinationAs_INT : I_INT;
	destinationAs_LINT : I_LINT;
	destinationAs_LREAL : I_LREAL;
	destinationAs_LWORD : I_LWORD;
	destinationAs_REAL : I_REAL;
	destinationAs_SINT : I_SINT;
	destinationAs_STRING : I_STRING;
	destinationAs_TOD : I_TOD;
	destinationAs_UDINT : I_UDINT;
	destinationAs_UINT : I_UINT;
	destinationAs_ULINT : I_ULINT;
	destinationAs_USINT : I_USINT;
	destinationAs_WORD : I_WORD;
END_VAR
IF destination.TryResolveAs_BIT(destinationAs_BIT) AND_THEN TryConvert_BOOL_TO_BOOL(activeData, resultofBitConversion) THEN
	destinationAs_BIT.Value := resultOfBitConversion;
	TryConvertTo_ := TRUE;
	RETURN;
END_IF

IF destination.TryResolveAs_BOOL(destinationAs_BOOL) THEN
	TryConvertTo_ := TryConvert_BOOL_TO_BOOL(activeData, destinationAs_BOOL.Value);
	RETURN;
END_IF
		
IF destination.TryResolveAs_BYTE(destinationAs_BYTE) THEN
	TryConvertTo_ := TryConvert_BOOL_TO_BYTE(activeData, destinationAs_BYTE.Value);
	RETURN;
END_IF

IF destination.TryResolveAs_DINT(destinationAs_DINT) THEN
	TryConvertTo_ := TryConvert_BOOL_TO_DINT(activeData, destinationAs_DINT.Value);
	RETURN;
END_IF

IF destination.TryResolveAs_DT(destinationAs_DT) THEN
	TryConvertTo_ := TryConvert_BOOL_TO_DT(activeData, destinationAs_DT.Value);
	RETURN;
END_IF

IF destination.TryResolveAs_DWORD(destinationAs_DWORD) THEN
	TryConvertTo_ := TryConvert_BOOL_TO_DWORD(activeData, destinationAs_DWORD.Value);
	RETURN;
END_IF

IF destination.TryResolveAs_INT(destinationAs_INT) THEN
	TryConvertTo_ := TryConvert_BOOL_TO_INT(activeData, destinationAs_INT.Value);
	RETURN;
END_IF

IF destination.TryResolveAs_LINT(destinationAs_LINT) THEN
	TryConvertTo_ := TryConvert_BOOL_TO_LINT(activeData, destinationAs_LINT.Value);
	RETURN;
END_IF

IF destination.TryResolveAs_LREAL(destinationAs_LREAL) THEN
	TryConvertTo_ := TryConvert_BOOL_TO_LREAL(activeData, destinationAs_LREAL.Value);
	RETURN;
END_IF

IF destination.TryResolveAs_LWORD(destinationAs_LWORD) THEN
	TryConvertTo_ := TryConvert_BOOL_TO_LWORD(activeData, destinationAs_LWORD.Value);
	RETURN;
END_IF

IF destination.TryResolveAs_REAL(destinationAs_REAL) THEN
	TryConvertTo_ := TryConvert_BOOL_TO_REAL(activeData, destinationAs_REAL.Value);
	RETURN;
END_IF

IF destination.TryResolveAs_SINT(destinationAs_SINT) THEN
	TryConvertTo_ := TryConvert_BOOL_TO_SINT(activeData, destinationAs_SINT.Value);
	RETURN;
END_IF

IF destination.TryResolveAs_STRING(destinationAs_STRING) THEN
	TryConvertTo_ := TryConvert_BOOL_TO_STRING(activeData, destinationAs_STRING.Value);
	RETURN;
END_IF

IF destination.TryResolveAs_TOD(destinationAs_TOD) THEN
	TryConvertTo_ := TryConvert_BOOL_TO_TOD(activeData, destinationAs_TOD.Value);
	RETURN;
END_IF

IF destination.TryResolveAs_UDINT(destinationAs_UDINT) THEN
	TryConvertTo_ := TryConvert_BOOL_TO_UDINT(activeData, destinationAs_UDINT.Value);
	RETURN;
END_IF

IF destination.TryResolveAs_UINT(destinationAs_UINT) THEN
	TryConvertTo_ := TryConvert_BOOL_TO_UINT(activeData, destinationAs_UINT.Value);
	RETURN;
END_IF

IF destination.TryResolveAs_ULINT(destinationAs_ULINT) THEN
	TryConvertTo_ := TryConvert_BOOL_TO_ULINT(activeData, destinationAs_ULINT.Value);
	RETURN;
END_IF

IF destination.TryResolveAs_USINT(destinationAs_USINT) THEN
	TryConvertTo_ := TryConvert_BOOL_TO_USINT(activeData, destinationAs_USINT.Value);
	RETURN;
END_IF

IF destination.TryResolveAs_WORD(destinationAs_WORD) THEN
	TryConvertTo_ := TryConvert_BOOL_TO_WORD(activeData, destinationAs_WORD.Value);
	RETURN;
END_IF
END_METHOD

METHOD TryDeserializeFrom : BOOL
VAR_INPUT
	Deserializer : I_Deserializer;
	Feedback : I_DeserializerFeedback;
END_VAR
TryDeserializeFrom := Deserializer.TryGetBool(activeData, Feedback);
END_METHOD

METHOD TryMakeReferenceTo : BOOL
VAR_INPUT
	Target : I_Datatype;
END_VAR
VAR
	pTargetData : POINTER TO BOOL;
END_VAR
IF NOT IsEquivalentTo(Target) THEN
	RETURN;
END_IF

pTargetData := Target.Address;
activeData REF= pTargetData^;
TryMakeReferenceTo := TRUE;
END_METHOD

METHOD PUBLIC TryResolveAs_BOOL : BOOL
VAR_INPUT
	Destination : REFERENCE TO I_BOOL;
END_VAR
Destination := THIS^;
TryResolveAs_BOOL := TRUE;
END_METHOD

PROPERTY PUBLIC TypeName : T_MAXSTRING
GET
TypeName := 'BOOL';
END_GET
END_PROPERTY

{warning disable C5410}
PROPERTY PUBLIC Value : REFERENCE TO BOOL
{warning restore C5410}
GET
Value REF= activeData;
END_GET
END_PROPERTY

END_FUNCTION_BLOCK

// mobject-datatypes/_Internal/Datatype/DatatypeBase
{attribute 'linkalways'} 
{attribute 'no_explicit_call' := 'This FB is a CLASS and must be accessed using methods or properties'}
{attribute 'enable_dynamic_creation'}
FUNCTION_BLOCK ABSTRACT DatatypeBase EXTENDS Disposable IMPLEMENTS I_Datatype
VAR
END_VAR

METHOD PROTECTED OnSerializeTypeWith
VAR_INPUT
	Serializer : I_Serializer;
END_VAR
Serializer.AddKeyString('typeName',TypeName);
END_METHOD

METHOD PUBLIC Accept
VAR_INPUT
	Visitor : I_DatatypeVisitor;
END_VAR
Visitor.VisitDatatype(this^);
END_METHOD

PROPERTY PUBLIC ABSTRACT Address : PVOID
GET
END_GET
END_PROPERTY

METHOD PUBLIC ABSTRACT ClearReference
VAR_INPUT
END_VAR
END_METHOD

METHOD PUBLIC ABSTRACT Clone : I_Datatype
END_METHOD

METHOD PUBLIC IsEquivalentTo : BOOL
VAR_INPUT
	Datatype : I_Datatype;
END_VAR
IF Datatype.Root.TypeName <> TypeName THEN
	RETURN;
END_IF

IF Datatype.Root.Size <> Size THEN
	RETURN;
END_IF

IsEquivalentTo := TRUE;
END_METHOD

PROPERTY PUBLIC IsNull : BOOL
GET
IsNull := FALSE;
END_GET
END_PROPERTY

PROPERTY PUBLIC IsUserDefined : BOOL
GET
IsUserDefined := FALSE;
END_GET
END_PROPERTY

PROPERTY PUBLIC Root : I_Datatype
GET
Root := this^;
END_GET
END_PROPERTY

METHOD PUBLIC SerializeTypeWith
VAR_INPUT
	Serializer : I_Serializer;
END_VAR
Serializer.StartObject();
OnSerializeTypeWith(Serializer);
Serializer.EndObject();
END_METHOD

METHOD PUBLIC ABSTRACT SerializeWith
VAR_INPUT
	Serializer : I_Serializer;
END_VAR
END_METHOD

PROPERTY PUBLIC ABSTRACT Size : UDINT
GET
END_GET
END_PROPERTY

METHOD PUBLIC TryConvertTo : BOOL
VAR_INPUT
	Destination : ANY;
END_VAR
TryConvertTo := FALSE;
END_METHOD

METHOD PUBLIC TryConvertTo_ : BOOL
VAR_INPUT
	Destination : I_Datatype;
END_VAR
TryConvertTo_ := FALSE;
END_METHOD

METHOD PUBLIC TryCopyFrom : BOOL
VAR_INPUT
	Source : I_Datatype;
END_VAR
IF NOT IsEquivalentTo(Source) THEN
	RETURN;
END_IF

memcpy(Address, Source.Address, Size);
TryCopyFrom := TRUE;
END_METHOD

METHOD PUBLIC ABSTRACT TryDeserializeFrom : BOOL
VAR_INPUT
	Deserializer : I_Deserializer;
	Feedback : I_DeserializerFeedback;
END_VAR
END_METHOD

METHOD PUBLIC ABSTRACT TryMakeReferenceTo : BOOL
VAR_INPUT
	Target : I_Datatype;
END_VAR
END_METHOD

METHOD PUBLIC TryResolveAs_ANY : BOOL
VAR_INPUT
	Destination : REFERENCE TO I_ANY;
END_VAR
TryResolveAs_ANY := FALSE;
END_METHOD

METHOD PUBLIC TryResolveAs_BIT : BOOL
VAR_INPUT
	Destination : REFERENCE TO I_BIT;
END_VAR
TryResolveAs_BIT := FALSE;
END_METHOD

METHOD PUBLIC TryResolveAs_BOOL : BOOL
VAR_INPUT
	Destination : REFERENCE TO I_BOOL;
END_VAR
TryResolveAs_BOOL := FALSE;
END_METHOD

METHOD PUBLIC TryResolveAs_BYTE : BOOL
VAR_INPUT
	Destination : REFERENCE TO I_BYTE;
END_VAR
TryResolveAs_BYTE := FALSE;
END_METHOD

METHOD PUBLIC TryResolveAs_DINT : BOOL
VAR_INPUT
	Destination : REFERENCE TO I_DINT;
END_VAR
TryResolveAs_DINT := FALSE;
END_METHOD

METHOD PUBLIC TryResolveAs_DT : BOOL
VAR_INPUT
	Destination : REFERENCE TO I_DT;
END_VAR
TryResolveAs_DT := FALSE;
END_METHOD

METHOD PUBLIC TryResolveAs_DWORD : BOOL
VAR_INPUT
	Destination : REFERENCE TO I_DWORD;
END_VAR
TryResolveAs_DWORD := FALSE;
END_METHOD

METHOD PUBLIC TryResolveAs_INT : BOOL
VAR_INPUT
	Destination : REFERENCE TO I_INT;
END_VAR
TryResolveAs_INT := FALSE;
END_METHOD

METHOD PUBLIC TryResolveAs_LINT : BOOL
VAR_INPUT
	Destination : REFERENCE TO I_LINT;
END_VAR
TryResolveAs_LINT := FALSE;
END_METHOD

METHOD PUBLIC TryResolveAs_LREAL : BOOL
VAR_INPUT
	Destination : REFERENCE TO I_LREAL;
END_VAR
TryResolveAs_LREAL := FALSE;
END_METHOD

METHOD PUBLIC TryResolveAs_LWORD : BOOL
VAR_INPUT
	Destination : REFERENCE TO I_LWORD;
END_VAR
TryResolveAs_LWORD := FALSE;
END_METHOD

METHOD PUBLIC TryResolveAs_PVOID : BOOL
VAR_INPUT
	Destination : REFERENCE TO I_PVOID;
END_VAR
TryResolveAs_PVOID := FALSE;
END_METHOD

METHOD PUBLIC TryResolveAs_REAL : BOOL
VAR_INPUT
	Destination : REFERENCE TO I_REAL;
END_VAR
TryResolveAs_REAL := FALSE;
END_METHOD

METHOD PUBLIC TryResolveAs_REFERENCE_TO : BOOL
VAR_INPUT
	Destination : REFERENCE TO I_REFERENCE_TO;
END_VAR
TryResolveAs_REFERENCE_TO := FALSE;
END_METHOD

METHOD PUBLIC TryResolveAs_SINT : BOOL
VAR_INPUT
	Destination : REFERENCE TO I_SINT;
END_VAR
TryResolveAs_SINT := FALSE;
END_METHOD

METHOD PUBLIC TryResolveAs_STRING : BOOL
VAR_INPUT
	Destination : REFERENCE TO I_STRING;
END_VAR
TryResolveAs_STRING := FALSE;
END_METHOD

METHOD PUBLIC TryResolveAs_TIME_OF_DAY : BOOL
VAR_INPUT
	Destination : REFERENCE TO I_TIME_OF_DAY;
END_VAR
TryResolveAs_TIME_OF_DAY := FALSE;
END_METHOD

METHOD PUBLIC TryResolveAs_TOD : BOOL
VAR_INPUT
	Destination : REFERENCE TO I_TOD;
END_VAR
TryResolveAs_TOD := FALSE;
END_METHOD

METHOD PUBLIC TryResolveAs_UDINT : BOOL
VAR_INPUT
	Destination : REFERENCE TO I_UDINT;
END_VAR
TryResolveAs_UDINT := FALSE;
END_METHOD

METHOD PUBLIC TryResolveAs_UINT : BOOL
VAR_INPUT
	Destination : REFERENCE TO I_UINT;
END_VAR
TryResolveAs_UINT := FALSE;
END_METHOD

METHOD PUBLIC TryResolveAs_ULINT : BOOL
VAR_INPUT
	Destination : REFERENCE TO I_ULINT;
END_VAR
TryResolveAs_ULINT := FALSE;
END_METHOD

METHOD PUBLIC TryResolveAs_USINT : BOOL
VAR_INPUT
	Destination : REFERENCE TO I_USINT;
END_VAR
TryResolveAs_USINT := FALSE;
END_METHOD

METHOD PUBLIC TryResolveAs_WORD : BOOL
VAR_INPUT
	Destination : REFERENCE TO I_WORD;
END_VAR
TryResolveAs_WORD := FALSE;
END_METHOD

METHOD PUBLIC TryResolveAsAliasDatatype : BOOL
VAR_INPUT
	Destination : REFERENCE TO I_AliasDatatype;
END_VAR
TryResolveAsAliasDatatype := FALSE;
END_METHOD

METHOD PUBLIC TryResolveAsArrayDatatype : BOOL
VAR_INPUT
	Destination : REFERENCE TO I_ArrayDatatype;
END_VAR
TryResolveAsArrayDatatype := FALSE;
END_METHOD

METHOD PUBLIC TryResolveAsBitDatatype : BOOL
VAR_INPUT
	Destination : REFERENCE TO I_BIT;
END_VAR
TryResolveAsBitDatatype := FALSE;
END_METHOD

METHOD PUBLIC TryResolveAsEnumDatatype : BOOL
VAR_INPUT
	Destination : REFERENCE TO I_EnumDatatype;
END_VAR
TryResolveAsEnumDatatype := FALSE;
END_METHOD

METHOD PUBLIC TryResolveAsInterfaceDatatype : BOOL
VAR_INPUT
	Destination : REFERENCE TO I_InterfaceDatatype;
END_VAR
TryResolveAsInterfaceDatatype := FALSE;
END_METHOD

METHOD PUBLIC TryResolveAsStructuredDatatype : BOOL
VAR_INPUT
	Destination : REFERENCE TO I_StructuredDatatype;
END_VAR
TryResolveAsStructuredDatatype := FALSE;
END_METHOD

METHOD PUBLIC TryResolveAsUserDefinedDatatype : BOOL
VAR_INPUT
	Destination : REFERENCE TO I_UserDefinedDatatype;
END_VAR
TryResolveAsUserDefinedDatatype := FALSE;
END_METHOD

PROPERTY PUBLIC ABSTRACT TypeName : T_MAXSTRING
GET
END_GET
END_PROPERTY

END_FUNCTION_BLOCK

// mobject-datatypes/_Internal/Datatype/Interface/I_Datatype
INTERFACE I_Datatype extends I_Serializable, I_Deserializable, I_Disposable

METHOD PUBLIC Accept
VAR_INPUT
	Visitor : I_DatatypeVisitor;
END_VAR
END_METHOD

PROPERTY PUBLIC Address : PVOID
GET
END_GET
END_PROPERTY

METHOD PUBLIC ClearReference
VAR_INPUT
END_VAR
END_METHOD

METHOD Clone : I_Datatype
END_METHOD

METHOD PUBLIC IsEquivalentTo : BOOL
VAR_INPUT
	Datatype : I_Datatype;
END_VAR
END_METHOD

PROPERTY PUBLIC IsNull : BOOL
GET
END_GET
END_PROPERTY

PROPERTY PUBLIC IsUserDefined : BOOL
GET
END_GET
END_PROPERTY

PROPERTY PUBLIC Root : I_Datatype
GET
END_GET
END_PROPERTY

METHOD PUBLIC SerializeTypeWith
VAR_INPUT
	Serializer : I_Serializer;
END_VAR
END_METHOD

PROPERTY PUBLIC Size : UDINT
GET
END_GET
END_PROPERTY

METHOD PUBLIC TryConvertTo : BOOL
VAR_INPUT
	Destination : ANY;
END_VAR
END_METHOD

METHOD PUBLIC TryConvertTo_ : BOOL
VAR_INPUT
	Destination : I_Datatype;
END_VAR
END_METHOD

METHOD PUBLIC TryCopyFrom : BOOL
VAR_INPUT
	Source : I_Datatype;
END_VAR
END_METHOD

